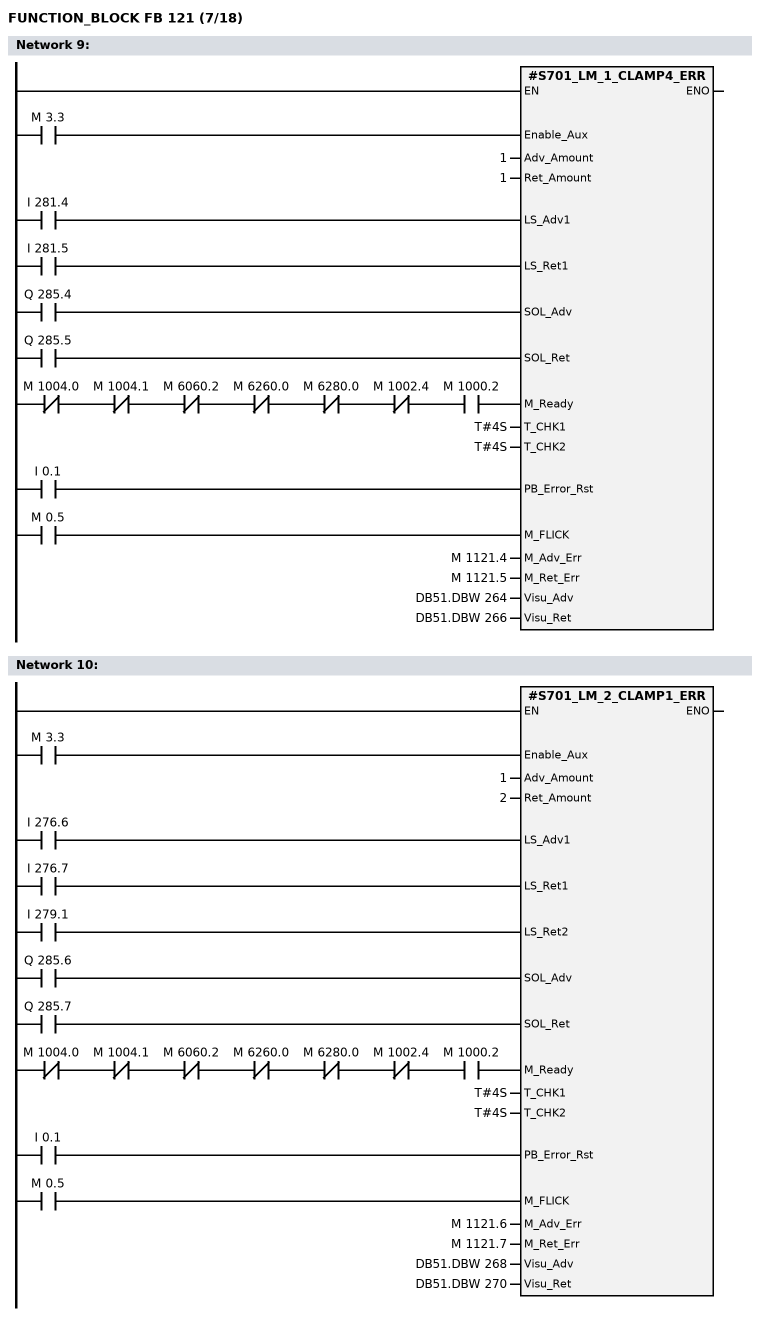

      A     M      3.3;
      =     L      0.0;
      BLD   103;
      A     I    281.4;
      =     L      0.1;
      BLD   103;
      A     I    281.5;
      =     L      0.2;
      BLD   103;
      A     Q    285.4;
      =     L      1.1;
      BLD   103;
      A     Q    285.5;
      =     L      1.2;
      BLD   103;
      AN    M   1004.0;
      AN    M   1004.1;
      AN    M   6060.2;
      AN    M   6260.0;
      AN    M   6280.0;
      AN    M   1002.4;
      A     M   1000.2;
      =     L      1.3;
      BLD   103;
      A     I      0.1;
      =     L      1.5;
      BLD   103;
      A     M      0.5;
      =     L      1.6;
      BLD   103;
      CALL #S701_LM_1_CLAMP4_ERR (
           Enable_Aux               := L      0.0,
           Adv_Amount               := 1,
           Ret_Amount               := 1,
           LS_Adv1                  := L      0.1,
           LS_Ret1                  := L      0.2,
           SOL_Adv                  := L      1.1,
           SOL_Ret                  := L      1.2,
           M_Ready                  := L      1.3,
           T_CHK1                   := T#4S,
           T_CHK2                   := T#4S,
           PB_Error_Rst             := L      1.5,
           M_FLICK                  := L      1.6,
           M_Adv_Err                := M   1121.4,
           M_Ret_Err                := M   1121.5,
           Visu_Adv                 := DB51.DBW  264,
           Visu_Ret                 := DB51.DBW  266);
      NOP   0;
NETWORK
TITLE =

      A     M      3.3;
      =     L      0.0;
      BLD   103;
      A     I    276.6;
      =     L      0.1;
      BLD   103;
      A     I    276.7;
      =     L      0.2;
      BLD   103;
      A     I    279.1;
      =     L      0.4;
      BLD   103;
      A     Q    285.6;
      =     L      1.1;
      BLD   103;
      A     Q    285.7;
      =     L      1.2;
      BLD   103;
      AN    M   1004.0;
      AN    M   1004.1;
      AN    M   6060.2;
      AN    M   6260.0;
      AN    M   6280.0;
      AN    M   1002.4;
      A     M   1000.2;
      =     L      1.3;
      BLD   103;
      A     I      0.1;
      =     L      1.5;
      BLD   103;
      A     M      0.5;
      =     L      1.6;
      BLD   103;
      CALL #S701_LM_2_CLAMP1_ERR (
           Enable_Aux               := L      0.0,
           Adv_Amount               := 1,
           Ret_Amount               := 2,
           LS_Adv1                  := L      0.1,
           LS_Ret1                  := L      0.2,
           LS_Ret2                  := L      0.4,
           SOL_Adv                  := L      1.1,
           SOL_Ret                  := L      1.2,
           M_Ready                  := L      1.3,
           T_CHK1                   := T#4S,
           T_CHK2                   := T#4S,
           PB_Error_Rst             := L      1.5,
           M_FLICK                  := L      1.6,
           M_Adv_Err                := M   1121.6,
           M_Ret_Err                := M   1121.7,
           Visu_Adv                 := DB51.DBW  268,
           Visu_Ret                 := DB51.DBW  270);
      NOP   0;
NETWORK
TITLE =
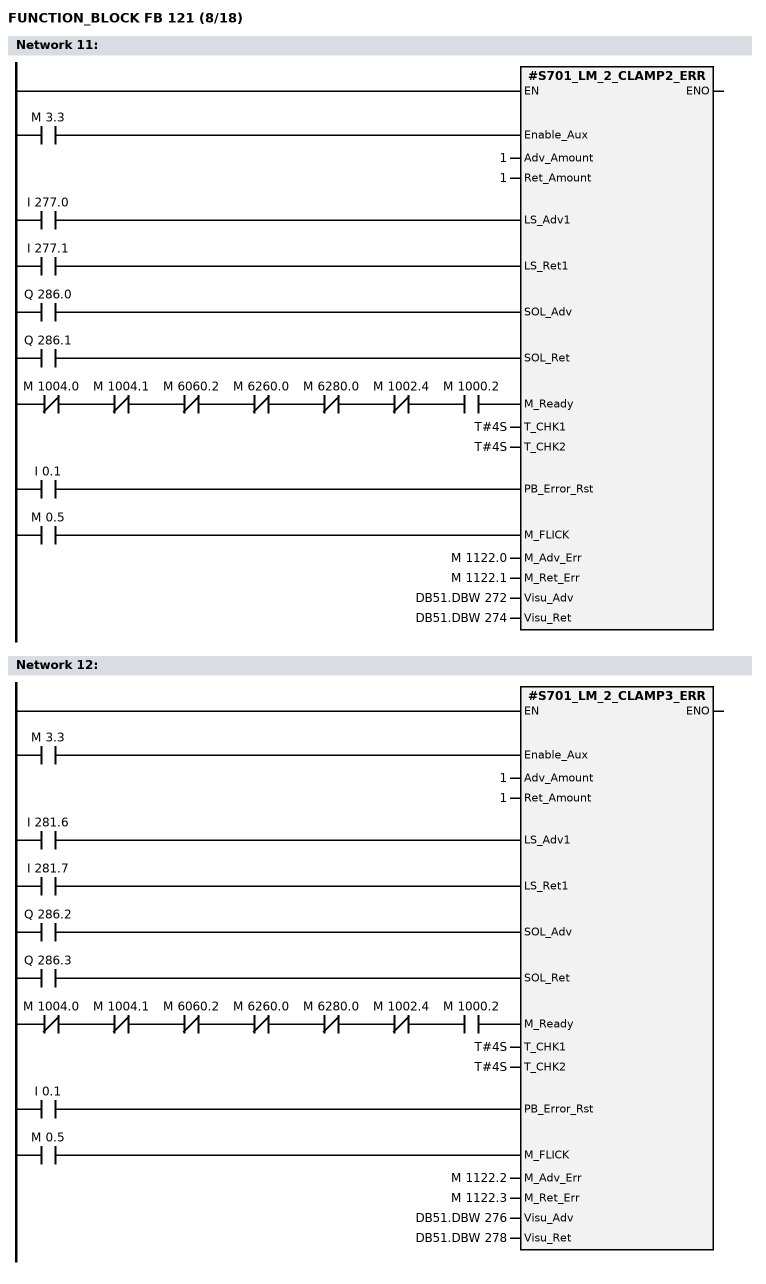

      A     M      3.3;
      =     L      0.0;
      BLD   103;
      A     I    277.0;
      =     L      0.1;
      BLD   103;
      A     I    277.1;
      =     L      0.2;
      BLD   103;
      A     Q    286.0;
      =     L      1.1;
      BLD   103;
      A     Q    286.1;
      =     L      1.2;
      BLD   103;
      AN    M   1004.0;
      AN    M   1004.1;
      AN    M   6060.2;
      AN    M   6260.0;
      AN    M   6280.0;
      AN    M   1002.4;
      A     M   1000.2;
      =     L      1.3;
      BLD   103;
      A     I      0.1;
      =     L      1.5;
      BLD   103;
      A     M      0.5;
      =     L      1.6;
      BLD   103;
      CALL #S701_LM_2_CLAMP2_ERR (
           Enable_Aux               := L      0.0,
           Adv_Amount               := 1,
           Ret_Amount               := 1,
           LS_Adv1                  := L      0.1,
           LS_Ret1                  := L      0.2,
           SOL_Adv                  := L      1.1,
           SOL_Ret                  := L      1.2,
           M_Ready                  := L      1.3,
           T_CHK1                   := T#4S,
           T_CHK2                   := T#4S,
           PB_Error_Rst             := L      1.5,
           M_FLICK                  := L      1.6,
           M_Adv_Err                := M   1122.0,
           M_Ret_Err                := M   1122.1,
           Visu_Adv                 := DB51.DBW  272,
           Visu_Ret                 := DB51.DBW  274);
      NOP   0;
NETWORK
TITLE =

      A     M      3.3;
      =     L      0.0;
      BLD   103;
      A     I    281.6;
      =     L      0.1;
      BLD   103;
      A     I    281.7;
      =     L      0.2;
      BLD   103;
      A     Q    286.2;
      =     L      1.1;
      BLD   103;
      A     Q    286.3;
      =     L      1.2;
      BLD   103;
      AN    M   1004.0;
      AN    M   1004.1;
      AN    M   6060.2;
      AN    M   6260.0;
      AN    M   6280.0;
      AN    M   1002.4;
      A     M   1000.2;
      =     L      1.3;
      BLD   103;
      A     I      0.1;
      =     L      1.5;
      BLD   103;
      A     M      0.5;
      =     L      1.6;
      BLD   103;
      CALL #S701_LM_2_CLAMP3_ERR (
           Enable_Aux               := L      0.0,
           Adv_Amount               := 1,
           Ret_Amount               := 1,
           LS_Adv1                  := L      0.1,
           LS_Ret1                  := L      0.2,
           SOL_Adv                  := L      1.1,
           SOL_Ret                  := L      1.2,
           M_Ready                  := L      1.3,
           T_CHK1                   := T#4S,
           T_CHK2                   := T#4S,
           PB_Error_Rst             := L      1.5,
           M_FLICK                  := L      1.6,
           M_Adv_Err                := M   1122.2,
           M_Ret_Err                := M   1122.3,
           Visu_Adv                 := DB51.DBW  276,
           Visu_Ret                 := DB51.DBW  278);
      NOP   0;
NETWORK
TITLE =
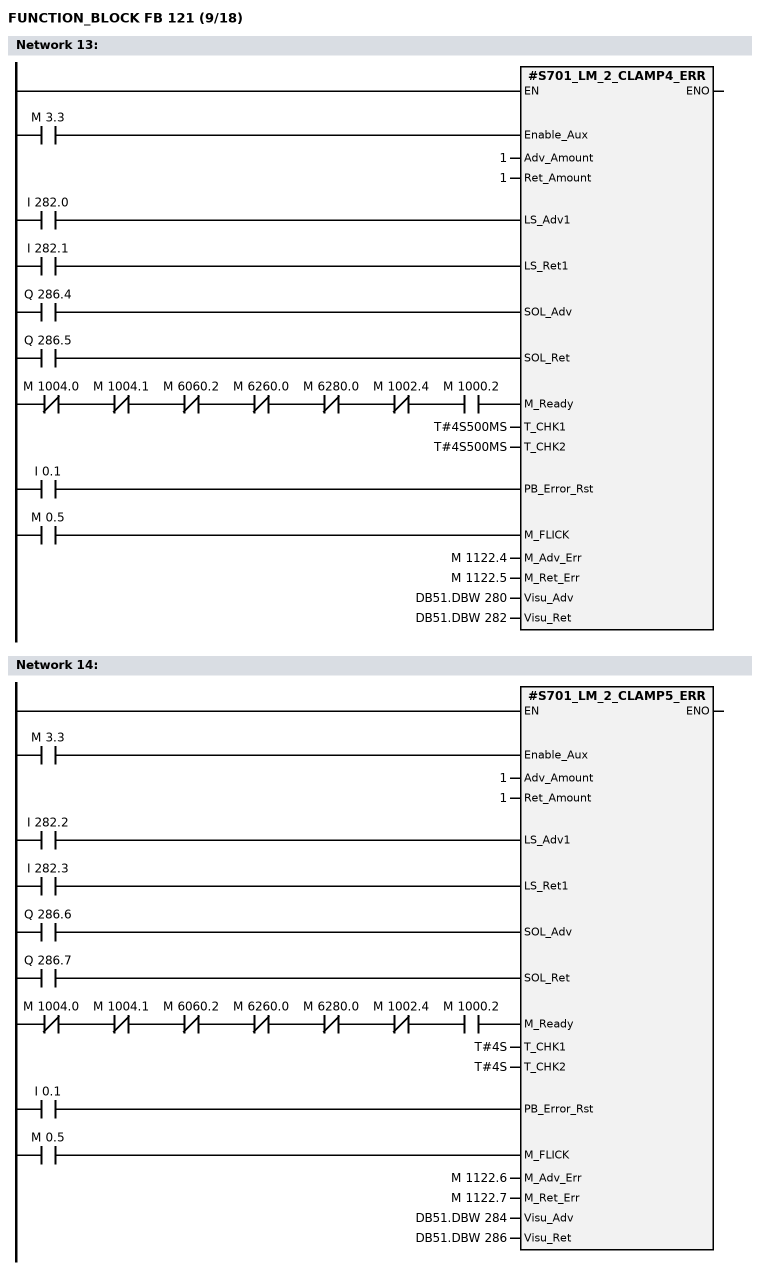

      A     M      3.3;
      =     L      0.0;
      BLD   103;
      A     I    282.0;
      =     L      0.1;
      BLD   103;
      A     I    282.1;
      =     L      0.2;
      BLD   103;
      A     Q    286.4;
      =     L      1.1;
      BLD   103;
      A     Q    286.5;
      =     L      1.2;
      BLD   103;
      AN    M   1004.0;
      AN    M   1004.1;
      AN    M   6060.2;
      AN    M   6260.0;
      AN    M   6280.0;
      AN    M   1002.4;
      A     M   1000.2;
      =     L      1.3;
      BLD   103;
      A     I      0.1;
      =     L      1.5;
      BLD   103;
      A     M      0.5;
      =     L      1.6;
      BLD   103;
      CALL #S701_LM_2_CLAMP4_ERR (
           Enable_Aux               := L      0.0,
           Adv_Amount               := 1,
           Ret_Amount               := 1,
           LS_Adv1                  := L      0.1,
           LS_Ret1                  := L      0.2,
           SOL_Adv                  := L      1.1,
           SOL_Ret                  := L      1.2,
           M_Ready                  := L      1.3,
           T_CHK1                   := T#4S500MS,
           T_CHK2                   := T#4S500MS,
           PB_Error_Rst             := L      1.5,
           M_FLICK                  := L      1.6,
           M_Adv_Err                := M   1122.4,
           M_Ret_Err                := M   1122.5,
           Visu_Adv                 := DB51.DBW  280,
           Visu_Ret                 := DB51.DBW  282);
      NOP   0;
NETWORK
TITLE =

      A     M      3.3;
      =     L      0.0;
      BLD   103;
      A     I    282.2;
      =     L      0.1;
      BLD   103;
      A     I    282.3;
      =     L      0.2;
      BLD   103;
      A     Q    286.6;
      =     L      1.1;
      BLD   103;
      A     Q    286.7;
      =     L      1.2;
      BLD   103;
      AN    M   1004.0;
      AN    M   1004.1;
      AN    M   6060.2;
      AN    M   6260.0;
      AN    M   6280.0;
      AN    M   1002.4;
      A     M   1000.2;
      =     L      1.3;
      BLD   103;
      A     I      0.1;
      =     L      1.5;
      BLD   103;
      A     M      0.5;
      =     L      1.6;
      BLD   103;
      CALL #S701_LM_2_CLAMP5_ERR (
           Enable_Aux               := L      0.0,
           Adv_Amount               := 1,
           Ret_Amount               := 1,
           LS_Adv1                  := L      0.1,
           LS_Ret1                  := L      0.2,
           SOL_Adv                  := L      1.1,
           SOL_Ret                  := L      1.2,
           M_Ready                  := L      1.3,
           T_CHK1                   := T#4S,
           T_CHK2                   := T#4S,
           PB_Error_Rst             := L      1.5,
           M_FLICK                  := L      1.6,
           M_Adv_Err                := M   1122.6,
           M_Ret_Err                := M   1122.7,
           Visu_Adv                 := DB51.DBW  284,
           Visu_Ret                 := DB51.DBW  286);
      NOP   0;
NETWORK
TITLE =
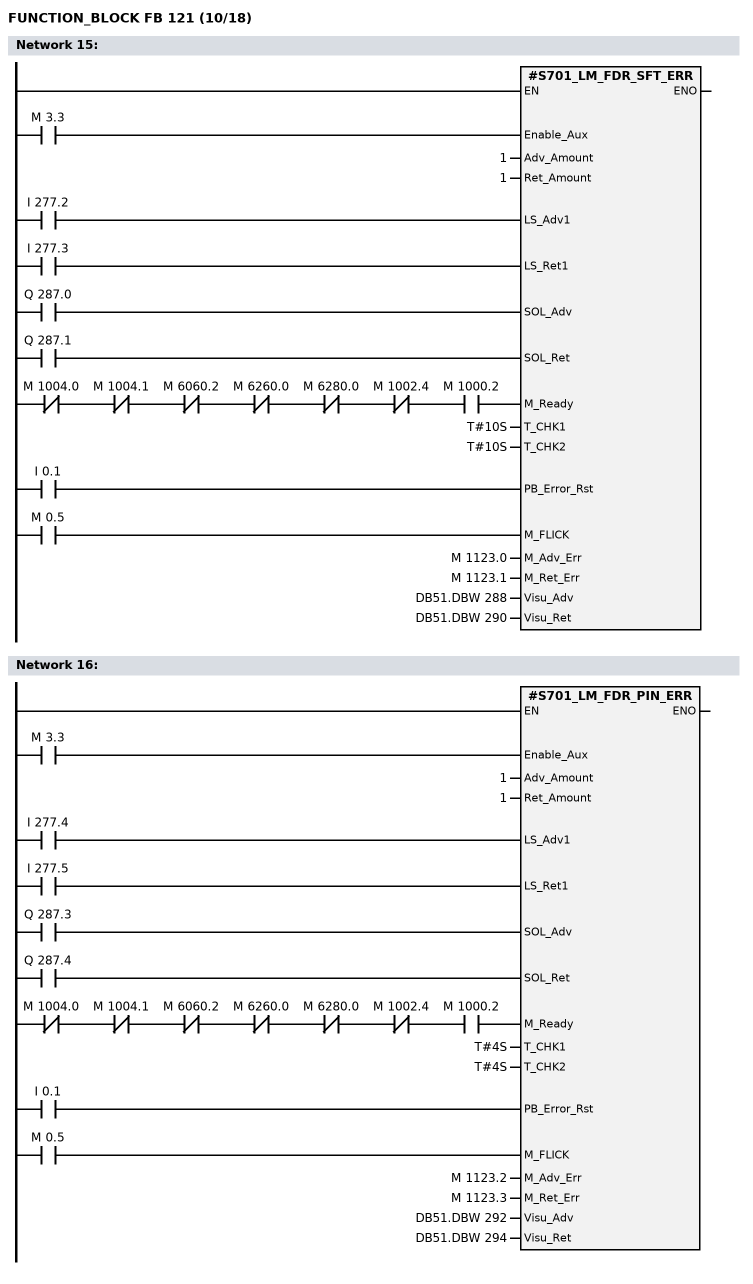

      A     M      3.3;
      =     L      0.0;
      BLD   103;
      A     I    277.2;
      =     L      0.1;
      BLD   103;
      A     I    277.3;
      =     L      0.2;
      BLD   103;
      A     Q    287.0;
      =     L      1.1;
      BLD   103;
      A     Q    287.1;
      =     L      1.2;
      BLD   103;
      AN    M   1004.0;
      AN    M   1004.1;
      AN    M   6060.2;
      AN    M   6260.0;
      AN    M   6280.0;
      AN    M   1002.4;
      A     M   1000.2;
      =     L      1.3;
      BLD   103;
      A     I      0.1;
      =     L      1.5;
      BLD   103;
      A     M      0.5;
      =     L      1.6;
      BLD   103;
      CALL #S701_LM_FDR_SFT_ERR (
           Enable_Aux               := L      0.0,
           Adv_Amount               := 1,
           Ret_Amount               := 1,
           LS_Adv1                  := L      0.1,
           LS_Ret1                  := L      0.2,
           SOL_Adv                  := L      1.1,
           SOL_Ret                  := L      1.2,
           M_Ready                  := L      1.3,
           T_CHK1                   := T#10S,
           T_CHK2                   := T#10S,
           PB_Error_Rst             := L      1.5,
           M_FLICK                  := L      1.6,
           M_Adv_Err                := M   1123.0,
           M_Ret_Err                := M   1123.1,
           Visu_Adv                 := DB51.DBW  288,
           Visu_Ret                 := DB51.DBW  290);
      NOP   0;
NETWORK
TITLE =

      A     M      3.3;
      =     L      0.0;
      BLD   103;
      A     I    277.4;
      =     L      0.1;
      BLD   103;
      A     I    277.5;
      =     L      0.2;
      BLD   103;
      A     Q    287.3;
      =     L      1.1;
      BLD   103;
      A     Q    287.4;
      =     L      1.2;
      BLD   103;
      AN    M   1004.0;
      AN    M   1004.1;
      AN    M   6060.2;
      AN    M   6260.0;
      AN    M   6280.0;
      AN    M   1002.4;
      A     M   1000.2;
      =     L      1.3;
      BLD   103;
      A     I      0.1;
      =     L      1.5;
      BLD   103;
      A     M      0.5;
      =     L      1.6;
      BLD   103;
      CALL #S701_LM_FDR_PIN_ERR (
           Enable_Aux               := L      0.0,
           Adv_Amount               := 1,
           Ret_Amount               := 1,
           LS_Adv1                  := L      0.1,
           LS_Ret1                  := L      0.2,
           SOL_Adv                  := L      1.1,
           SOL_Ret                  := L      1.2,
           M_Ready                  := L      1.3,
           T_CHK1                   := T#4S,
           T_CHK2                   := T#4S,
           PB_Error_Rst             := L      1.5,
           M_FLICK                  := L      1.6,
           M_Adv_Err                := M   1123.2,
           M_Ret_Err                := M   1123.3,
           Visu_Adv                 := DB51.DBW  292,
           Visu_Ret                 := DB51.DBW  294);
      NOP   0;
NETWORK
TITLE =
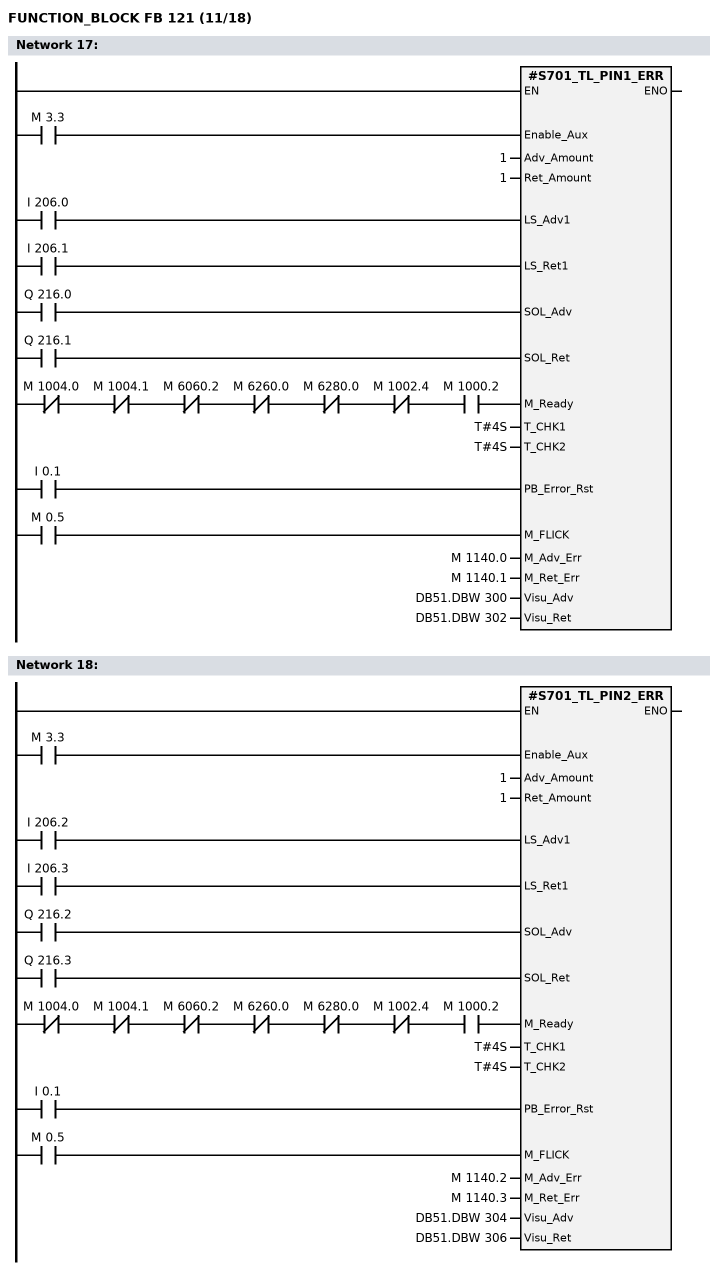

      A     M      3.3;
      =     L      0.0;
      BLD   103;
      A     I    206.0;
      =     L      0.1;
      BLD   103;
      A     I    206.1;
      =     L      0.2;
      BLD   103;
      A     Q    216.0;
      =     L      1.1;
      BLD   103;
      A     Q    216.1;
      =     L      1.2;
      BLD   103;
      AN    M   1004.0;
      AN    M   1004.1;
      AN    M   6060.2;
      AN    M   6260.0;
      AN    M   6280.0;
      AN    M   1002.4;
      A     M   1000.2;
      =     L      1.3;
      BLD   103;
      A     I      0.1;
      =     L      1.5;
      BLD   103;
      A     M      0.5;
      =     L      1.6;
      BLD   103;
      CALL #S701_TL_PIN1_ERR (
           Enable_Aux               := L      0.0,
           Adv_Amount               := 1,
           Ret_Amount               := 1,
           LS_Adv1                  := L      0.1,
           LS_Ret1                  := L      0.2,
           SOL_Adv                  := L      1.1,
           SOL_Ret                  := L      1.2,
           M_Ready                  := L      1.3,
           T_CHK1                   := T#4S,
           T_CHK2                   := T#4S,
           PB_Error_Rst             := L      1.5,
           M_FLICK                  := L      1.6,
           M_Adv_Err                := M   1140.0,
           M_Ret_Err                := M   1140.1,
           Visu_Adv                 := DB51.DBW  300,
           Visu_Ret                 := DB51.DBW  302);
      NOP   0;
NETWORK
TITLE =

      A     M      3.3;
      =     L      0.0;
      BLD   103;
      A     I    206.2;
      =     L      0.1;
      BLD   103;
      A     I    206.3;
      =     L      0.2;
      BLD   103;
      A     Q    216.2;
      =     L      1.1;
      BLD   103;
      A     Q    216.3;
      =     L      1.2;
      BLD   103;
      AN    M   1004.0;
      AN    M   1004.1;
      AN    M   6060.2;
      AN    M   6260.0;
      AN    M   6280.0;
      AN    M   1002.4;
      A     M   1000.2;
      =     L      1.3;
      BLD   103;
      A     I      0.1;
      =     L      1.5;
      BLD   103;
      A     M      0.5;
      =     L      1.6;
      BLD   103;
      CALL #S701_TL_PIN2_ERR (
           Enable_Aux               := L      0.0,
           Adv_Amount               := 1,
           Ret_Amount               := 1,
           LS_Adv1                  := L      0.1,
           LS_Ret1                  := L      0.2,
           SOL_Adv                  := L      1.1,
           SOL_Ret                  := L      1.2,
           M_Ready                  := L      1.3,
           T_CHK1                   := T#4S,
           T_CHK2                   := T#4S,
           PB_Error_Rst             := L      1.5,
           M_FLICK                  := L      1.6,
           M_Adv_Err                := M   1140.2,
           M_Ret_Err                := M   1140.3,
           Visu_Adv                 := DB51.DBW  304,
           Visu_Ret                 := DB51.DBW  306);
      NOP   0;
NETWORK
TITLE =
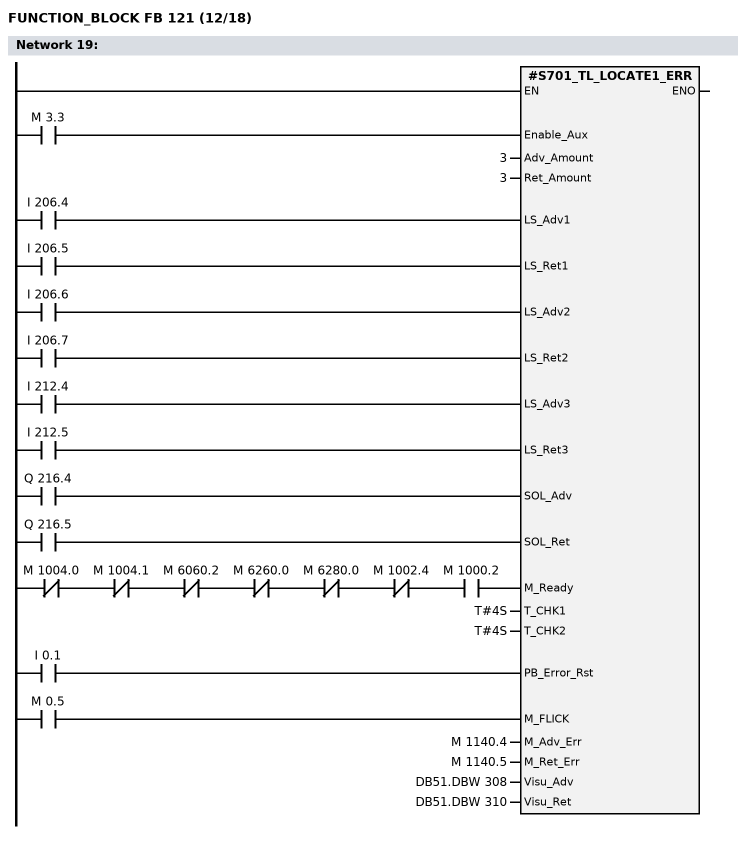

      A     M      3.3;
      =     L      0.0;
      BLD   103;
      A     I    206.4;
      =     L      0.1;
      BLD   103;
      A     I    206.5;
      =     L      0.2;
      BLD   103;
      A     I    206.6;
      =     L      0.3;
      BLD   103;
      A     I    206.7;
      =     L      0.4;
      BLD   103;
      A     I    212.4;
      =     L      0.5;
      BLD   103;
      A     I    212.5;
      =     L      0.6;
      BLD   103;
      A     Q    216.4;
      =     L      1.1;
      BLD   103;
      A     Q    216.5;
      =     L      1.2;
      BLD   103;
      AN    M   1004.0;
      AN    M   1004.1;
      AN    M   6060.2;
      AN    M   6260.0;
      AN    M   6280.0;
      AN    M   1002.4;
      A     M   1000.2;
      =     L      1.3;
      BLD   103;
      A     I      0.1;
      =     L      1.5;
      BLD   103;
      A     M      0.5;
      =     L      1.6;
      BLD   103;
      CALL #S701_TL_LOCATE1_ERR (
           Enable_Aux               := L      0.0,
           Adv_Amount               := 3,
           Ret_Amount               := 3,
           LS_Adv1                  := L      0.1,
           LS_Ret1                  := L      0.2,
           LS_Adv2                  := L      0.3,
           LS_Ret2                  := L      0.4,
           LS_Adv3                  := L      0.5,
           LS_Ret3                  := L      0.6,
           SOL_Adv                  := L      1.1,
           SOL_Ret                  := L      1.2,
           M_Ready                  := L      1.3,
           T_CHK1                   := T#4S,
           T_CHK2                   := T#4S,
           PB_Error_Rst             := L      1.5,
           M_FLICK                  := L      1.6,
           M_Adv_Err                := M   1140.4,
           M_Ret_Err                := M   1140.5,
           Visu_Adv                 := DB51.DBW  308,
           Visu_Ret                 := DB51.DBW  310);
      NOP   0;
NETWORK
TITLE =
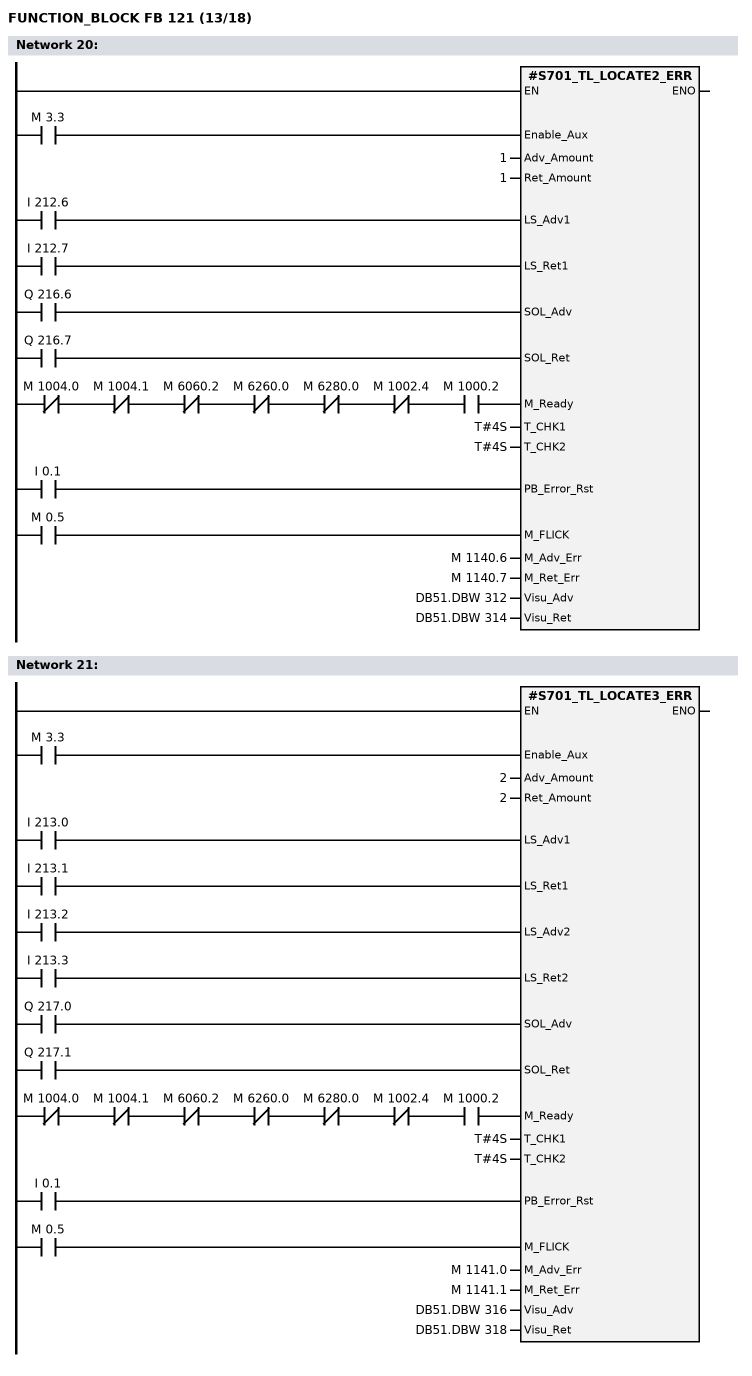

      A     M      3.3;
      =     L      0.0;
      BLD   103;
      A     I    212.6;
      =     L      0.1;
      BLD   103;
      A     I    212.7;
      =     L      0.2;
      BLD   103;
      A     Q    216.6;
      =     L      1.1;
      BLD   103;
      A     Q    216.7;
      =     L      1.2;
      BLD   103;
      AN    M   1004.0;
      AN    M   1004.1;
      AN    M   6060.2;
      AN    M   6260.0;
      AN    M   6280.0;
      AN    M   1002.4;
      A     M   1000.2;
      =     L      1.3;
      BLD   103;
      A     I      0.1;
      =     L      1.5;
      BLD   103;
      A     M      0.5;
      =     L      1.6;
      BLD   103;
      CALL #S701_TL_LOCATE2_ERR (
           Enable_Aux               := L      0.0,
           Adv_Amount               := 1,
           Ret_Amount               := 1,
           LS_Adv1                  := L      0.1,
           LS_Ret1                  := L      0.2,
           SOL_Adv                  := L      1.1,
           SOL_Ret                  := L      1.2,
           M_Ready                  := L      1.3,
           T_CHK1                   := T#4S,
           T_CHK2                   := T#4S,
           PB_Error_Rst             := L      1.5,
           M_FLICK                  := L      1.6,
           M_Adv_Err                := M   1140.6,
           M_Ret_Err                := M   1140.7,
           Visu_Adv                 := DB51.DBW  312,
           Visu_Ret                 := DB51.DBW  314);
      NOP   0;
NETWORK
TITLE =

      A     M      3.3;
      =     L      0.0;
      BLD   103;
      A     I    213.0;
      =     L      0.1;
      BLD   103;
      A     I    213.1;
      =     L      0.2;
      BLD   103;
      A     I    213.2;
      =     L      0.3;
      BLD   103;
      A     I    213.3;
      =     L      0.4;
      BLD   103;
      A     Q    217.0;
      =     L      1.1;
      BLD   103;
      A     Q    217.1;
      =     L      1.2;
      BLD   103;
      AN    M   1004.0;
      AN    M   1004.1;
      AN    M   6060.2;
      AN    M   6260.0;
      AN    M   6280.0;
      AN    M   1002.4;
      A     M   1000.2;
      =     L      1.3;
      BLD   103;
      A     I      0.1;
      =     L      1.5;
      BLD   103;
      A     M      0.5;
      =     L      1.6;
      BLD   103;
      CALL #S701_TL_LOCATE3_ERR (
           Enable_Aux               := L      0.0,
           Adv_Amount               := 2,
           Ret_Amount               := 2,
           LS_Adv1                  := L      0.1,
           LS_Ret1                  := L      0.2,
           LS_Adv2                  := L      0.3,
           LS_Ret2                  := L      0.4,
           SOL_Adv                  := L      1.1,
           SOL_Ret                  := L      1.2,
           M_Ready                  := L      1.3,
           T_CHK1                   := T#4S,
           T_CHK2                   := T#4S,
           PB_Error_Rst             := L      1.5,
           M_FLICK                  := L      1.6,
           M_Adv_Err                := M   1141.0,
           M_Ret_Err                := M   1141.1,
           Visu_Adv                 := DB51.DBW  316,
           Visu_Ret                 := DB51.DBW  318);
      NOP   0;
NETWORK
TITLE =
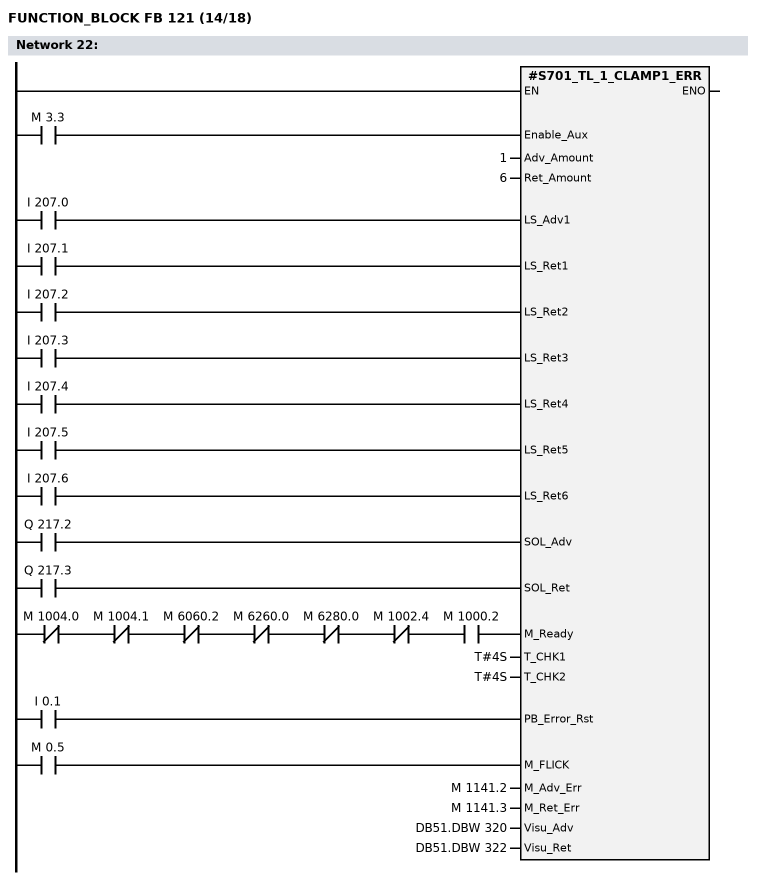

      A     M      3.3;
      =     L      0.0;
      BLD   103;
      A     I    207.0;
      =     L      0.1;
      BLD   103;
      A     I    207.1;
      =     L      0.2;
      BLD   103;
      A     I    207.2;
      =     L      0.4;
      BLD   103;
      A     I    207.3;
      =     L      0.6;
      BLD   103;
      A     I    207.4;
      =     L      1.0;
      BLD   103;
      A     I    207.5;
      =     L      1.2;
      BLD   103;
      A     I    207.6;
      =     L      1.4;
      BLD   103;
      A     Q    217.2;
      =     L      2.1;
      BLD   103;
      A     Q    217.3;
      =     L      2.2;
      BLD   103;
      AN    M   1004.0;
      AN    M   1004.1;
      AN    M   6060.2;
      AN    M   6260.0;
      AN    M   6280.0;
      AN    M   1002.4;
      A     M   1000.2;
      =     L      2.3;
      BLD   103;
      A     I      0.1;
      =     L      2.5;
      BLD   103;
      A     M      0.5;
      =     L      2.6;
      BLD   103;
      CALL #S701_TL_1_CLAMP1_ERR (
           Enable_Aux               := L      0.0,
           Adv_Amount               := 1,
           Ret_Amount               := 6,
           LS_Adv1                  := L      0.1,
           LS_Ret1                  := L      0.2,
           LS_Ret2                  := L      0.4,
           LS_Ret3                  := L      0.6,
           LS_Ret4                  := L      1.0,
           LS_Ret5                  := L      1.2,
           LS_Ret6                  := L      1.4,
           SOL_Adv                  := L      2.1,
           SOL_Ret                  := L      2.2,
           M_Ready                  := L      2.3,
           T_CHK1                   := T#4S,
           T_CHK2                   := T#4S,
           PB_Error_Rst             := L      2.5,
           M_FLICK                  := L      2.6,
           M_Adv_Err                := M   1141.2,
           M_Ret_Err                := M   1141.3,
           Visu_Adv                 := DB51.DBW  320,
           Visu_Ret                 := DB51.DBW  322);
      NOP   0;
NETWORK
TITLE =
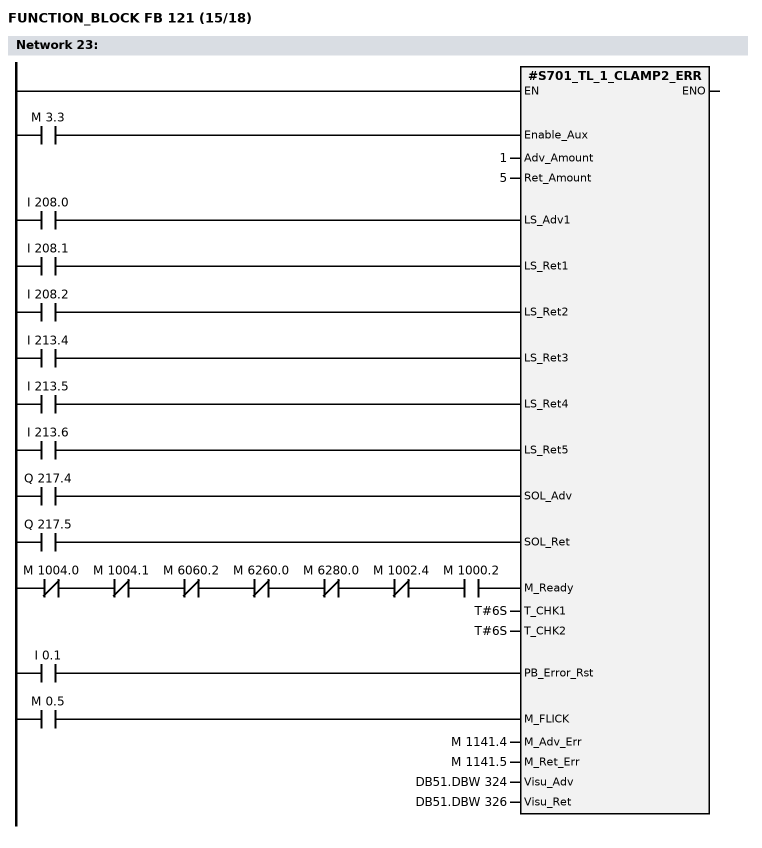

      A     M      3.3;
      =     L      0.0;
      BLD   103;
      A     I    208.0;
      =     L      0.1;
      BLD   103;
      A     I    208.1;
      =     L      0.2;
      BLD   103;
      A     I    208.2;
      =     L      0.4;
      BLD   103;
      A     I    213.4;
      =     L      0.6;
      BLD   103;
      A     I    213.5;
      =     L      1.0;
      BLD   103;
      A     I    213.6;
      =     L      1.2;
      BLD   103;
      A     Q    217.4;
      =     L      2.1;
      BLD   103;
      A     Q    217.5;
      =     L      2.2;
      BLD   103;
      AN    M   1004.0;
      AN    M   1004.1;
      AN    M   6060.2;
      AN    M   6260.0;
      AN    M   6280.0;
      AN    M   1002.4;
      A     M   1000.2;
      =     L      2.3;
      BLD   103;
      A     I      0.1;
      =     L      2.5;
      BLD   103;
      A     M      0.5;
      =     L      2.6;
      BLD   103;
      CALL #S701_TL_1_CLAMP2_ERR (
           Enable_Aux               := L      0.0,
           Adv_Amount               := 1,
           Ret_Amount               := 5,
           LS_Adv1                  := L      0.1,
           LS_Ret1                  := L      0.2,
           LS_Ret2                  := L      0.4,
           LS_Ret3                  := L      0.6,
           LS_Ret4                  := L      1.0,
           LS_Ret5                  := L      1.2,
           SOL_Adv                  := L      2.1,
           SOL_Ret                  := L      2.2,
           M_Ready                  := L      2.3,
           T_CHK1                   := T#6S,
           T_CHK2                   := T#6S,
           PB_Error_Rst             := L      2.5,
           M_FLICK                  := L      2.6,
           M_Adv_Err                := M   1141.4,
           M_Ret_Err                := M   1141.5,
           Visu_Adv                 := DB51.DBW  324,
           Visu_Ret                 := DB51.DBW  326);
      NOP   0;
NETWORK
TITLE =
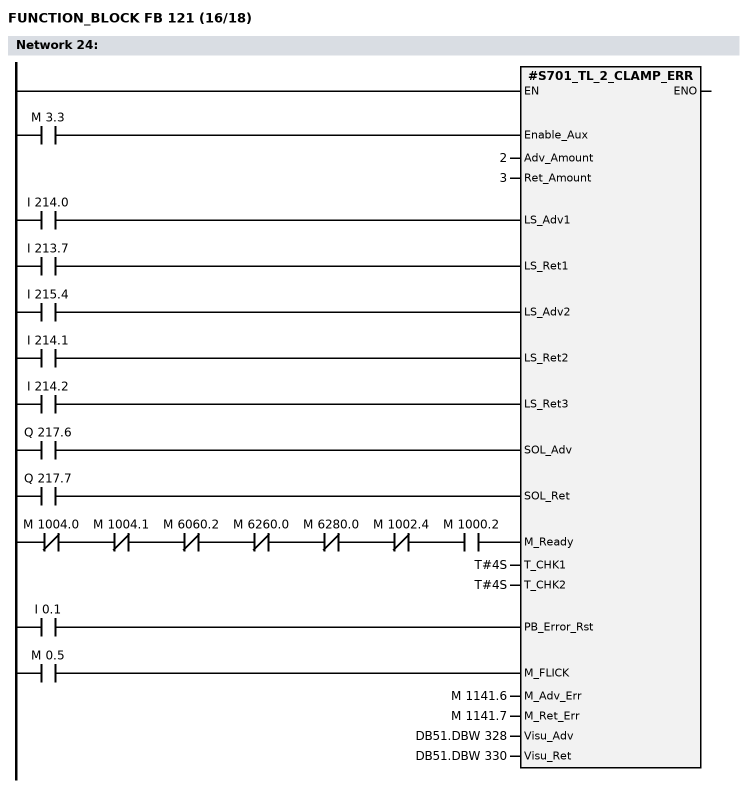

      A     M      3.3;
      =     L      0.0;
      BLD   103;
      A     I    214.0;
      =     L      0.1;
      BLD   103;
      A     I    213.7;
      =     L      0.2;
      BLD   103;
      A     I    215.4;
      =     L      0.3;
      BLD   103;
      A     I    214.1;
      =     L      0.4;
      BLD   103;
      A     I    214.2;
      =     L      0.6;
      BLD   103;
      A     Q    217.6;
      =     L      2.1;
      BLD   103;
      A     Q    217.7;
      =     L      2.2;
      BLD   103;
      AN    M   1004.0;
      AN    M   1004.1;
      AN    M   6060.2;
      AN    M   6260.0;
      AN    M   6280.0;
      AN    M   1002.4;
      A     M   1000.2;
      =     L      2.3;
      BLD   103;
      A     I      0.1;
      =     L      2.5;
      BLD   103;
      A     M      0.5;
      =     L      2.6;
      BLD   103;
      CALL #S701_TL_2_CLAMP_ERR (
           Enable_Aux               := L      0.0,
           Adv_Amount               := 2,
           Ret_Amount               := 3,
           LS_Adv1                  := L      0.1,
           LS_Ret1                  := L      0.2,
           LS_Adv2                  := L      0.3,
           LS_Ret2                  := L      0.4,
           LS_Ret3                  := L      0.6,
           SOL_Adv                  := L      2.1,
           SOL_Ret                  := L      2.2,
           M_Ready                  := L      2.3,
           T_CHK1                   := T#4S,
           T_CHK2                   := T#4S,
           PB_Error_Rst             := L      2.5,
           M_FLICK                  := L      2.6,
           M_Adv_Err                := M   1141.6,
           M_Ret_Err                := M   1141.7,
           Visu_Adv                 := DB51.DBW  328,
           Visu_Ret                 := DB51.DBW  330);
      NOP   0;
NETWORK
TITLE =
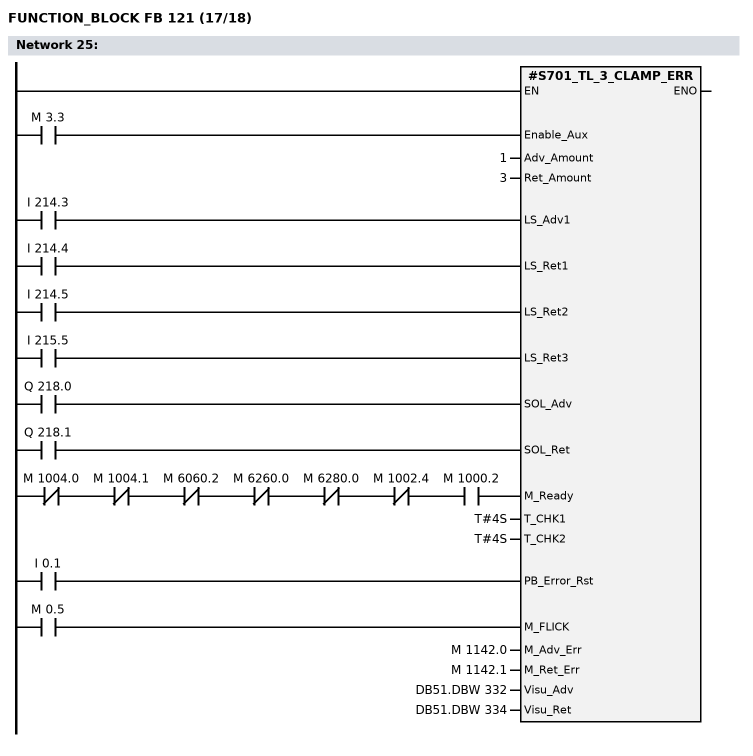

      A     M      3.3;
      =     L      0.0;
      BLD   103;
      A     I    214.3;
      =     L      0.1;
      BLD   103;
      A     I    214.4;
      =     L      0.2;
      BLD   103;
      A     I    214.5;
      =     L      0.4;
      BLD   103;
      A     I    215.5;
      =     L      0.6;
      BLD   103;
      A     Q    218.0;
      =     L      2.1;
      BLD   103;
      A     Q    218.1;
      =     L      2.2;
      BLD   103;
      AN    M   1004.0;
      AN    M   1004.1;
      AN    M   6060.2;
      AN    M   6260.0;
      AN    M   6280.0;
      AN    M   1002.4;
      A     M   1000.2;
      =     L      2.3;
      BLD   103;
      A     I      0.1;
      =     L      2.5;
      BLD   103;
      A     M      0.5;
      =     L      2.6;
      BLD   103;
      CALL #S701_TL_3_CLAMP_ERR (
           Enable_Aux               := L      0.0,
           Adv_Amount               := 1,
           Ret_Amount               := 3,
           LS_Adv1                  := L      0.1,
           LS_Ret1                  := L      0.2,
           LS_Ret2                  := L      0.4,
           LS_Ret3                  := L      0.6,
           SOL_Adv                  := L      2.1,
           SOL_Ret                  := L      2.2,
           M_Ready                  := L      2.3,
           T_CHK1                   := T#4S,
           T_CHK2                   := T#4S,
           PB_Error_Rst             := L      2.5,
           M_FLICK                  := L      2.6,
           M_Adv_Err                := M   1142.0,
           M_Ret_Err                := M   1142.1,
           Visu_Adv                 := DB51.DBW  332,
           Visu_Ret                 := DB51.DBW  334);
      NOP   0;
NETWORK
TITLE =
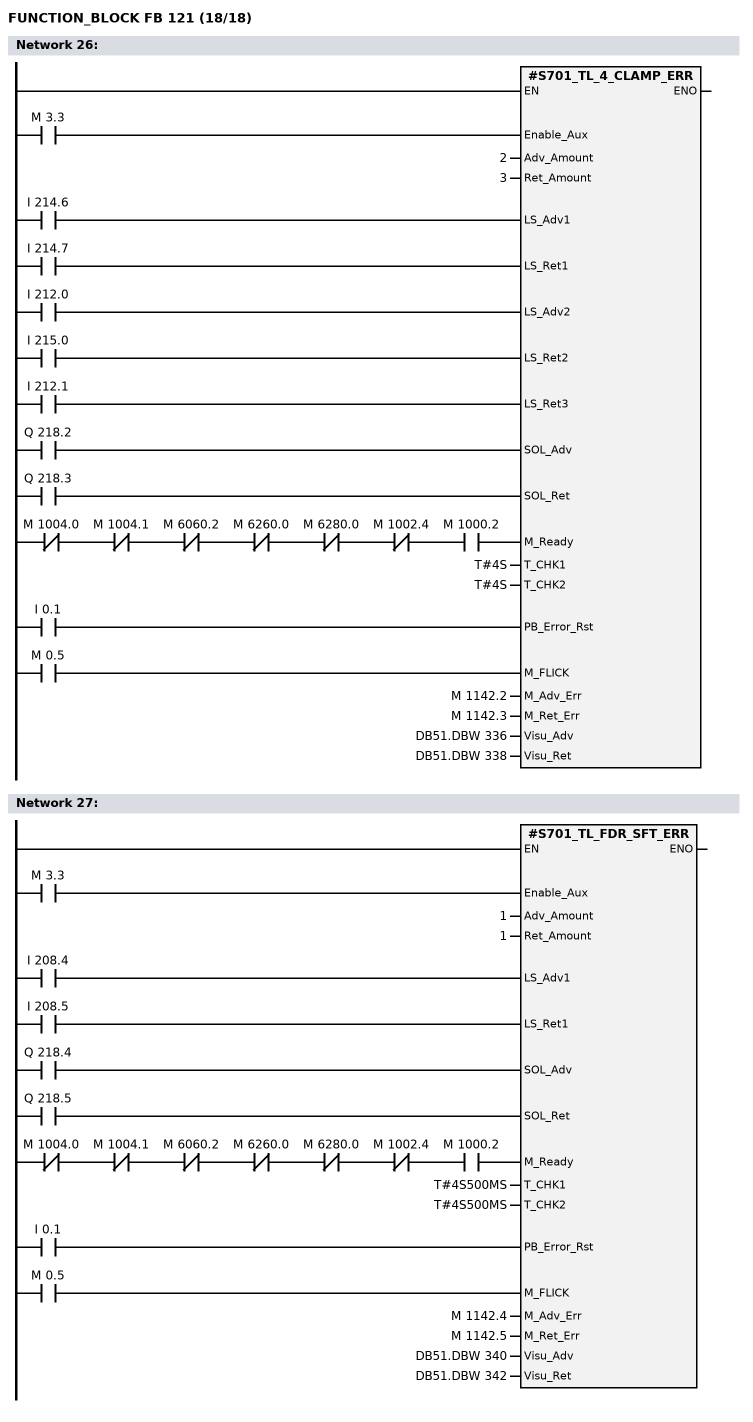

      A     M      3.3;
      =     L      0.0;
      BLD   103;
      A     I    214.6;
      =     L      0.1;
      BLD   103;
      A     I    214.7;
      =     L      0.2;
      BLD   103;
      A     I    212.0;
      =     L      0.3;
      BLD   103;
      A     I    215.0;
      =     L      0.4;
      BLD   103;
      A     I    212.1;
      =     L      0.6;
      BLD   103;
      A     Q    218.2;
      =     L      2.1;
      BLD   103;
      A     Q    218.3;
      =     L      2.2;
      BLD   103;
      AN    M   1004.0;
      AN    M   1004.1;
      AN    M   6060.2;
      AN    M   6260.0;
      AN    M   6280.0;
      AN    M   1002.4;
      A     M   1000.2;
      =     L      2.3;
      BLD   103;
      A     I      0.1;
      =     L      2.5;
      BLD   103;
      A     M      0.5;
      =     L      2.6;
      BLD   103;
      CALL #S701_TL_4_CLAMP_ERR (
           Enable_Aux               := L      0.0,
           Adv_Amount               := 2,
           Ret_Amount               := 3,
           LS_Adv1                  := L      0.1,
           LS_Ret1                  := L      0.2,
           LS_Adv2                  := L      0.3,
           LS_Ret2                  := L      0.4,
           LS_Ret3                  := L      0.6,
           SOL_Adv                  := L      2.1,
           SOL_Ret                  := L      2.2,
           M_Ready                  := L      2.3,
           T_CHK1                   := T#4S,
           T_CHK2                   := T#4S,
           PB_Error_Rst             := L      2.5,
           M_FLICK                  := L      2.6,
           M_Adv_Err                := M   1142.2,
           M_Ret_Err                := M   1142.3,
           Visu_Adv                 := DB51.DBW  336,
           Visu_Ret                 := DB51.DBW  338);
      NOP   0;
NETWORK
TITLE =

      A     M      3.3;
      =     L      0.0;
      BLD   103;
      A     I    208.4;
      =     L      0.1;
      BLD   103;
      A     I    208.5;
      =     L      0.2;
      BLD   103;
      A     Q    218.4;
      =     L      2.1;
      BLD   103;
      A     Q    218.5;
      =     L      2.2;
      BLD   103;
      AN    M   1004.0;
      AN    M   1004.1;
      AN    M   6060.2;
      AN    M   6260.0;
      AN    M   6280.0;
      AN    M   1002.4;
      A     M   1000.2;
      =     L      2.3;
      BLD   103;
      A     I      0.1;
      =     L      2.5;
      BLD   103;
      A     M      0.5;
      =     L      2.6;
      BLD   103;
      CALL #S701_TL_FDR_SFT_ERR (
           Enable_Aux               := L      0.0,
           Adv_Amount               := 1,
           Ret_Amount               := 1,
           LS_Adv1                  := L      0.1,
           LS_Ret1                  := L      0.2,
           SOL_Adv                  := L      2.1,
           SOL_Ret                  := L      2.2,
           M_Ready                  := L      2.3,
           T_CHK1                   := T#4S500MS,
           T_CHK2                   := T#4S500MS,
           PB_Error_Rst             := L      2.5,
           M_FLICK                  := L      2.6,
           M_Adv_Err                := M   1142.4,
           M_Ret_Err                := M   1142.5,
           Visu_Adv                 := DB51.DBW  340,
           Visu_Ret                 := DB51.DBW  342);
      NOP   0;
END_FUNCTION_BLOCK

DATA_BLOCK DB 121
TITLE =
VERSION : 0.0

 FB 121
BEGIN
   S701_RETURN_LOCK_ERR.Enable_Aux := FALSE;
   S701_RETURN_LOCK_ERR.Adv_Amount := 0;
   S701_RETURN_LOCK_ERR.Ret_Amount := 0;
   S701_RETURN_LOCK_ERR.LS_Adv1 := FALSE;
   S701_RETURN_LOCK_ERR.LS_Ret1 := FALSE;
   S701_RETURN_LOCK_ERR.LS_Adv2 := FALSE;
   S701_RETURN_LOCK_ERR.LS_Ret2 := FALSE;
   S701_RETURN_LOCK_ERR.LS_Adv3 := FALSE;
   S701_RETURN_LOCK_ERR.LS_Ret3 := FALSE;
   S701_RETURN_LOCK_ERR.LS_Adv4 := FALSE;
   S701_RETURN_LOCK_ERR.LS_Ret4 := FALSE;
   S701_RETURN_LOCK_ERR.SOL_Adv := FALSE;
   S701_RETURN_LOCK_ERR.SOL_Ret := FALSE;
   S701_RETURN_LOCK_ERR.M_Ready := FALSE;
   S701_RETURN_LOCK_ERR.T_CHK1 := T#0MS;
   S701_RETURN_LOCK_ERR.T_CHK2 := T#0MS;
   S701_RETURN_LOCK_ERR.PB_Lamp_CHK := FALSE;
   S701_RETURN_LOCK_ERR.PB_Error_Rst := FALSE;
   S701_RETURN_LOCK_ERR.M_FLICK := FALSE;
   S701_RETURN_LOCK_ERR.M_Adv_Err := FALSE;
   S701_RETURN_LOCK_ERR.M_Ret_Err := FALSE;
   S701_RETURN_LOCK_ERR.LP_Adv := FALSE;
   S701_RETURN_LOCK_ERR.LP_Ret := FALSE;
   S701_RETURN_LOCK_ERR.Visu_Adv := W#16#0;
   S701_RETURN_LOCK_ERR.Visu_Ret := W#16#0;
   S701_RETURN_LOCK_ERR.Error_T1.IN := FALSE;
   S701_RETURN_LOCK_ERR.Error_T1.PT := T#0MS;
   S701_RETURN_LOCK_ERR.Error_T1.Q := FALSE;
   S701_RETURN_LOCK_ERR.Error_T1.ET := T#0MS;
   S701_RETURN_LOCK_ERR.Error_T1.STATE := B#16#0;
   S701_RETURN_LOCK_ERR.Error_T1.STIME := T#0MS;
   S701_RETURN_LOCK_ERR.Error_T1.ATIME := T#0MS;
   S701_RETURN_LOCK_ERR.Error_T2.IN := FALSE;
   S701_RETURN_LOCK_ERR.Error_T2.PT := T#0MS;
   S701_RETURN_LOCK_ERR.Error_T2.Q := FALSE;
   S701_RETURN_LOCK_ERR.Error_T2.ET := T#0MS;
   S701_RETURN_LOCK_ERR.Error_T2.STATE := B#16#0;
   S701_RETURN_LOCK_ERR.Error_T2.STIME := T#0MS;
   S701_RETURN_LOCK_ERR.Error_T2.ATIME := T#0MS;
   S701_RETURN_LOCK_ERR.CHK_Aux1 := FALSE;
   S701_RETURN_LOCK_ERR.CHK_Aux2 := FALSE;
   S701_RETURN_LOCK_ERR.Error_T1_DN := FALSE;
   S701_RETURN_LOCK_ERR.Error_T2_DN := FALSE;
   S701_RETURN_LOCK_ERR.Adv_Memo := FALSE;
   S701_RETURN_LOCK_ERR.Visu_Adv_Arr[0] := FALSE;
   S701_RETURN_LOCK_ERR.Visu_Adv_Arr[1] := FALSE;
   S701_RETURN_LOCK_ERR.Visu_Adv_Arr[2] := FALSE;
   S701_RETURN_LOCK_ERR.Visu_Adv_Arr[3] := FALSE;
   S701_RETURN_LOCK_ERR.Visu_Adv_Arr[4] := FALSE;
   S701_RETURN_LOCK_ERR.Visu_Adv_Arr[5] := FALSE;
   S701_RETURN_LOCK_ERR.Visu_Adv_Arr[6] := FALSE;
   S701_RETURN_LOCK_ERR.Visu_Adv_Arr[7] := FALSE;
   S701_RETURN_LOCK_ERR.Visu_Adv_Arr[8] := FALSE;
   S701_RETURN_LOCK_ERR.Visu_Adv_Arr[9] := FALSE;
   S701_RETURN_LOCK_ERR.Visu_Adv_Arr[10] := FALSE;
   S701_RETURN_LOCK_ERR.Visu_Adv_Arr[11] := FALSE;
   S701_RETURN_LOCK_ERR.Visu_Adv_Arr[12] := FALSE;
   S701_RETURN_LOCK_ERR.Visu_Adv_Arr[13] := FALSE;
   S701_RETURN_LOCK_ERR.Visu_Adv_Arr[14] := FALSE;
   S701_RETURN_LOCK_ERR.Visu_Adv_Arr[15] := FALSE;
   S701_RETURN_LOCK_ERR.Visu_Ret_Arr[0] := FALSE;
   S701_RETURN_LOCK_ERR.Visu_Ret_Arr[1] := FALSE;
   S701_RETURN_LOCK_ERR.Visu_Ret_Arr[2] := FALSE;
   S701_RETURN_LOCK_ERR.Visu_Ret_Arr[3] := FALSE;
   S701_RETURN_LOCK_ERR.Visu_Ret_Arr[4] := FALSE;
   S701_RETURN_LOCK_ERR.Visu_Ret_Arr[5] := FALSE;
   S701_RETURN_LOCK_ERR.Visu_Ret_Arr[6] := FALSE;
   S701_RETURN_LOCK_ERR.Visu_Ret_Arr[7] := FALSE;
   S701_RETURN_LOCK_ERR.Visu_Ret_Arr[8] := FALSE;
   S701_RETURN_LOCK_ERR.Visu_Ret_Arr[9] := FALSE;
   S701_RETURN_LOCK_ERR.Visu_Ret_Arr[10] := FALSE;
   S701_RETURN_LOCK_ERR.Visu_Ret_Arr[11] := FALSE;
   S701_RETURN_LOCK_ERR.Visu_Ret_Arr[12] := FALSE;
   S701_RETURN_LOCK_ERR.Visu_Ret_Arr[13] := FALSE;
   S701_RETURN_LOCK_ERR.Visu_Ret_Arr[14] := FALSE;
   S701_RETURN_LOCK_ERR.Visu_Ret_Arr[15] := FALSE;
   S701_RETURN_LOCK_ERR.BLK_Move_Ret := 0;
   S701_RETURN_LOCK_ERR.Enable := FALSE;
   S701_RETURN_LOCK_ERR.Adv_End := FALSE;
   S701_RETURN_LOCK_ERR.Ret_End := FALSE;
   S701_TURN_LOCK_ERR.Enable_Aux := FALSE;
   S701_TURN_LOCK_ERR.Adv_Amount := 0;
   S701_TURN_LOCK_ERR.Ret_Amount := 0;
   S701_TURN_LOCK_ERR.LS_Adv1 := FALSE;
   S701_TURN_LOCK_ERR.LS_Ret1 := FALSE;
   S701_TURN_LOCK_ERR.LS_Adv2 := FALSE;
   S701_TURN_LOCK_ERR.LS_Ret2 := FALSE;
   S701_TURN_LOCK_ERR.LS_Adv3 := FALSE;
   S701_TURN_LOCK_ERR.LS_Ret3 := FALSE;
   S701_TURN_LOCK_ERR.LS_Adv4 := FALSE;
   S701_TURN_LOCK_ERR.LS_Ret4 := FALSE;
   S701_TURN_LOCK_ERR.SOL_Adv := FALSE;
   S701_TURN_LOCK_ERR.SOL_Ret := FALSE;
   S701_TURN_LOCK_ERR.M_Ready := FALSE;
   S701_TURN_LOCK_ERR.T_CHK1 := T#0MS;
   S701_TURN_LOCK_ERR.T_CHK2 := T#0MS;
   S701_TURN_LOCK_ERR.PB_Lamp_CHK := FALSE;
   S701_TURN_LOCK_ERR.PB_Error_Rst := FALSE;
   S701_TURN_LOCK_ERR.M_FLICK := FALSE;
   S701_TURN_LOCK_ERR.M_Adv_Err := FALSE;
   S701_TURN_LOCK_ERR.M_Ret_Err := FALSE;
   S701_TURN_LOCK_ERR.LP_Adv := FALSE;
   S701_TURN_LOCK_ERR.LP_Ret := FALSE;
   S701_TURN_LOCK_ERR.Visu_Adv := W#16#0;
   S701_TURN_LOCK_ERR.Visu_Ret := W#16#0;
   S701_TURN_LOCK_ERR.Error_T1.IN := FALSE;
   S701_TURN_LOCK_ERR.Error_T1.PT := T#0MS;
   S701_TURN_LOCK_ERR.Error_T1.Q := FALSE;
   S701_TURN_LOCK_ERR.Error_T1.ET := T#0MS;
   S701_TURN_LOCK_ERR.Error_T1.STATE := B#16#0;
   S701_TURN_LOCK_ERR.Error_T1.STIME := T#0MS;
   S701_TURN_LOCK_ERR.Error_T1.ATIME := T#0MS;
   S701_TURN_LOCK_ERR.Error_T2.IN := FALSE;
   S701_TURN_LOCK_ERR.Error_T2.PT := T#0MS;
   S701_TURN_LOCK_ERR.Error_T2.Q := FALSE;
   S701_TURN_LOCK_ERR.Error_T2.ET := T#0MS;
   S701_TURN_LOCK_ERR.Error_T2.STATE := B#16#0;
   S701_TURN_LOCK_ERR.Error_T2.STIME := T#0MS;
   S701_TURN_LOCK_ERR.Error_T2.ATIME := T#0MS;
   S701_TURN_LOCK_ERR.CHK_Aux1 := FALSE;
   S701_TURN_LOCK_ERR.CHK_Aux2 := FALSE;
   S701_TURN_LOCK_ERR.Error_T1_DN := FALSE;
   S701_TURN_LOCK_ERR.Error_T2_DN := FALSE;
   S701_TURN_LOCK_ERR.Adv_Memo := FALSE;
   S701_TURN_LOCK_ERR.Visu_Adv_Arr[0] := FALSE;
   S701_TURN_LOCK_ERR.Visu_Adv_Arr[1] := FALSE;
   S701_TURN_LOCK_ERR.Visu_Adv_Arr[2] := FALSE;
   S701_TURN_LOCK_ERR.Visu_Adv_Arr[3] := FALSE;
   S701_TURN_LOCK_ERR.Visu_Adv_Arr[4] := FALSE;
   S701_TURN_LOCK_ERR.Visu_Adv_Arr[5] := FALSE;
   S701_TURN_LOCK_ERR.Visu_Adv_Arr[6] := FALSE;
   S701_TURN_LOCK_ERR.Visu_Adv_Arr[7] := FALSE;
   S701_TURN_LOCK_ERR.Visu_Adv_Arr[8] := FALSE;
   S701_TURN_LOCK_ERR.Visu_Adv_Arr[9] := FALSE;
   S701_TURN_LOCK_ERR.Visu_Adv_Arr[10] := FALSE;
   S701_TURN_LOCK_ERR.Visu_Adv_Arr[11] := FALSE;
   S701_TURN_LOCK_ERR.Visu_Adv_Arr[12] := FALSE;
   S701_TURN_LOCK_ERR.Visu_Adv_Arr[13] := FALSE;
   S701_TURN_LOCK_ERR.Visu_Adv_Arr[14] := FALSE;
   S701_TURN_LOCK_ERR.Visu_Adv_Arr[15] := FALSE;
   S701_TURN_LOCK_ERR.Visu_Ret_Arr[0] := FALSE;
   S701_TURN_LOCK_ERR.Visu_Ret_Arr[1] := FALSE;
   S701_TURN_LOCK_ERR.Visu_Ret_Arr[2] := FALSE;
   S701_TURN_LOCK_ERR.Visu_Ret_Arr[3] := FALSE;
   S701_TURN_LOCK_ERR.Visu_Ret_Arr[4] := FALSE;
   S701_TURN_LOCK_ERR.Visu_Ret_Arr[5] := FALSE;
   S701_TURN_LOCK_ERR.Visu_Ret_Arr[6] := FALSE;
   S701_TURN_LOCK_ERR.Visu_Ret_Arr[7] := FALSE;
   S701_TURN_LOCK_ERR.Visu_Ret_Arr[8] := FALSE;
   S701_TURN_LOCK_ERR.Visu_Ret_Arr[9] := FALSE;
   S701_TURN_LOCK_ERR.Visu_Ret_Arr[10] := FALSE;
   S701_TURN_LOCK_ERR.Visu_Ret_Arr[11] := FALSE;
   S701_TURN_LOCK_ERR.Visu_Ret_Arr[12] := FALSE;
   S701_TURN_LOCK_ERR.Visu_Ret_Arr[13] := FALSE;
   S701_TURN_LOCK_ERR.Visu_Ret_Arr[14] := FALSE;
   S701_TURN_LOCK_ERR.Visu_Ret_Arr[15] := FALSE;
   S701_TURN_LOCK_ERR.BLK_Move_Ret := 0;
   S701_TURN_LOCK_ERR.Enable := FALSE;
   S701_TURN_LOCK_ERR.Adv_End := FALSE;
   S701_TURN_LOCK_ERR.Ret_End := FALSE;
   S701_LM_PIN1_ERR.Enable_Aux := FALSE;
   S701_LM_PIN1_ERR.Adv_Amount := 0;
   S701_LM_PIN1_ERR.Ret_Amount := 0;
   S701_LM_PIN1_ERR.LS_Adv1 := FALSE;
   S701_LM_PIN1_ERR.LS_Ret1 := FALSE;
   S701_LM_PIN1_ERR.LS_Adv2 := FALSE;
   S701_LM_PIN1_ERR.LS_Ret2 := FALSE;
   S701_LM_PIN1_ERR.LS_Adv3 := FALSE;
   S701_LM_PIN1_ERR.LS_Ret3 := FALSE;
   S701_LM_PIN1_ERR.LS_Adv4 := FALSE;
   S701_LM_PIN1_ERR.LS_Ret4 := FALSE;
   S701_LM_PIN1_ERR.SOL_Adv := FALSE;
   S701_LM_PIN1_ERR.SOL_Ret := FALSE;
   S701_LM_PIN1_ERR.M_Ready := FALSE;
   S701_LM_PIN1_ERR.T_CHK1 := T#0MS;
   S701_LM_PIN1_ERR.T_CHK2 := T#0MS;
   S701_LM_PIN1_ERR.PB_Lamp_CHK := FALSE;
   S701_LM_PIN1_ERR.PB_Error_Rst := FALSE;
   S701_LM_PIN1_ERR.M_FLICK := FALSE;
   S701_LM_PIN1_ERR.M_Adv_Err := FALSE;
   S701_LM_PIN1_ERR.M_Ret_Err := FALSE;
   S701_LM_PIN1_ERR.LP_Adv := FALSE;
   S701_LM_PIN1_ERR.LP_Ret := FALSE;
   S701_LM_PIN1_ERR.Visu_Adv := W#16#0;
   S701_LM_PIN1_ERR.Visu_Ret := W#16#0;
   S701_LM_PIN1_ERR.Error_T1.IN := FALSE;
   S701_LM_PIN1_ERR.Error_T1.PT := T#0MS;
   S701_LM_PIN1_ERR.Error_T1.Q := FALSE;
   S701_LM_PIN1_ERR.Error_T1.ET := T#0MS;
   S701_LM_PIN1_ERR.Error_T1.STATE := B#16#0;
   S701_LM_PIN1_ERR.Error_T1.STIME := T#0MS;
   S701_LM_PIN1_ERR.Error_T1.ATIME := T#0MS;
   S701_LM_PIN1_ERR.Error_T2.IN := FALSE;
   S701_LM_PIN1_ERR.Error_T2.PT := T#0MS;
   S701_LM_PIN1_ERR.Error_T2.Q := FALSE;
   S701_LM_PIN1_ERR.Error_T2.ET := T#0MS;
   S701_LM_PIN1_ERR.Error_T2.STATE := B#16#0;
   S701_LM_PIN1_ERR.Error_T2.STIME := T#0MS;
   S701_LM_PIN1_ERR.Error_T2.ATIME := T#0MS;
   S701_LM_PIN1_ERR.CHK_Aux1 := FALSE;
   S701_LM_PIN1_ERR.CHK_Aux2 := FALSE;
   S701_LM_PIN1_ERR.Error_T1_DN := FALSE;
   S701_LM_PIN1_ERR.Error_T2_DN := FALSE;
   S701_LM_PIN1_ERR.Adv_Memo := FALSE;
   S701_LM_PIN1_ERR.Visu_Adv_Arr[0] := FALSE;
   S701_LM_PIN1_ERR.Visu_Adv_Arr[1] := FALSE;
   S701_LM_PIN1_ERR.Visu_Adv_Arr[2] := FALSE;
   S701_LM_PIN1_ERR.Visu_Adv_Arr[3] := FALSE;
   S701_LM_PIN1_ERR.Visu_Adv_Arr[4] := FALSE;
   S701_LM_PIN1_ERR.Visu_Adv_Arr[5] := FALSE;
   S701_LM_PIN1_ERR.Visu_Adv_Arr[6] := FALSE;
   S701_LM_PIN1_ERR.Visu_Adv_Arr[7] := FALSE;
   S701_LM_PIN1_ERR.Visu_Adv_Arr[8] := FALSE;
   S701_LM_PIN1_ERR.Visu_Adv_Arr[9] := FALSE;
   S701_LM_PIN1_ERR.Visu_Adv_Arr[10] := FALSE;
   S701_LM_PIN1_ERR.Visu_Adv_Arr[11] := FALSE;
   S701_LM_PIN1_ERR.Visu_Adv_Arr[12] := FALSE;
   S701_LM_PIN1_ERR.Visu_Adv_Arr[13] := FALSE;
   S701_LM_PIN1_ERR.Visu_Adv_Arr[14] := FALSE;
   S701_LM_PIN1_ERR.Visu_Adv_Arr[15] := FALSE;
   S701_LM_PIN1_ERR.Visu_Ret_Arr[0] := FALSE;
   S701_LM_PIN1_ERR.Visu_Ret_Arr[1] := FALSE;
   S701_LM_PIN1_ERR.Visu_Ret_Arr[2] := FALSE;
   S701_LM_PIN1_ERR.Visu_Ret_Arr[3] := FALSE;
   S701_LM_PIN1_ERR.Visu_Ret_Arr[4] := FALSE;
   S701_LM_PIN1_ERR.Visu_Ret_Arr[5] := FALSE;
   S701_LM_PIN1_ERR.Visu_Ret_Arr[6] := FALSE;
   S701_LM_PIN1_ERR.Visu_Ret_Arr[7] := FALSE;
   S701_LM_PIN1_ERR.Visu_Ret_Arr[8] := FALSE;
   S701_LM_PIN1_ERR.Visu_Ret_Arr[9] := FALSE;
   S701_LM_PIN1_ERR.Visu_Ret_Arr[10] := FALSE;
   S701_LM_PIN1_ERR.Visu_Ret_Arr[11] := FALSE;
   S701_LM_PIN1_ERR.Visu_Ret_Arr[12] := FALSE;
   S701_LM_PIN1_ERR.Visu_Ret_Arr[13] := FALSE;
   S701_LM_PIN1_ERR.Visu_Ret_Arr[14] := FALSE;
   S701_LM_PIN1_ERR.Visu_Ret_Arr[15] := FALSE;
   S701_LM_PIN1_ERR.BLK_Move_Ret := 0;
   S701_LM_PIN1_ERR.Enable := FALSE;
   S701_LM_PIN1_ERR.Adv_End := FALSE;
   S701_LM_PIN1_ERR.Ret_End := FALSE;
   S701_LM_PIN2_ERR.Enable_Aux := FALSE;
   S701_LM_PIN2_ERR.Adv_Amount := 0;
   S701_LM_PIN2_ERR.Ret_Amount := 0;
   S701_LM_PIN2_ERR.LS_Adv1 := FALSE;
   S701_LM_PIN2_ERR.LS_Ret1 := FALSE;
   S701_LM_PIN2_ERR.LS_Adv2 := FALSE;
   S701_LM_PIN2_ERR.LS_Ret2 := FALSE;
   S701_LM_PIN2_ERR.LS_Adv3 := FALSE;
   S701_LM_PIN2_ERR.LS_Ret3 := FALSE;
   S701_LM_PIN2_ERR.LS_Adv4 := FALSE;
   S701_LM_PIN2_ERR.LS_Ret4 := FALSE;
   S701_LM_PIN2_ERR.SOL_Adv := FALSE;
   S701_LM_PIN2_ERR.SOL_Ret := FALSE;
   S701_LM_PIN2_ERR.M_Ready := FALSE;
   S701_LM_PIN2_ERR.T_CHK1 := T#0MS;
   S701_LM_PIN2_ERR.T_CHK2 := T#0MS;
   S701_LM_PIN2_ERR.PB_Lamp_CHK := FALSE;
   S701_LM_PIN2_ERR.PB_Error_Rst := FALSE;
   S701_LM_PIN2_ERR.M_FLICK := FALSE;
   S701_LM_PIN2_ERR.M_Adv_Err := FALSE;
   S701_LM_PIN2_ERR.M_Ret_Err := FALSE;
   S701_LM_PIN2_ERR.LP_Adv := FALSE;
   S701_LM_PIN2_ERR.LP_Ret := FALSE;
   S701_LM_PIN2_ERR.Visu_Adv := W#16#0;
   S701_LM_PIN2_ERR.Visu_Ret := W#16#0;
   S701_LM_PIN2_ERR.Error_T1.IN := FALSE;
   S701_LM_PIN2_ERR.Error_T1.PT := T#0MS;
   S701_LM_PIN2_ERR.Error_T1.Q := FALSE;
   S701_LM_PIN2_ERR.Error_T1.ET := T#0MS;
   S701_LM_PIN2_ERR.Error_T1.STATE := B#16#0;
   S701_LM_PIN2_ERR.Error_T1.STIME := T#0MS;
   S701_LM_PIN2_ERR.Error_T1.ATIME := T#0MS;
   S701_LM_PIN2_ERR.Error_T2.IN := FALSE;
   S701_LM_PIN2_ERR.Error_T2.PT := T#0MS;
   S701_LM_PIN2_ERR.Error_T2.Q := FALSE;
   S701_LM_PIN2_ERR.Error_T2.ET := T#0MS;
   S701_LM_PIN2_ERR.Error_T2.STATE := B#16#0;
   S701_LM_PIN2_ERR.Error_T2.STIME := T#0MS;
   S701_LM_PIN2_ERR.Error_T2.ATIME := T#0MS;
   S701_LM_PIN2_ERR.CHK_Aux1 := FALSE;
   S701_LM_PIN2_ERR.CHK_Aux2 := FALSE;
   S701_LM_PIN2_ERR.Error_T1_DN := FALSE;
   S701_LM_PIN2_ERR.Error_T2_DN := FALSE;
   S701_LM_PIN2_ERR.Adv_Memo := FALSE;
   S701_LM_PIN2_ERR.Visu_Adv_Arr[0] := FALSE;
   S701_LM_PIN2_ERR.Visu_Adv_Arr[1] := FALSE;
   S701_LM_PIN2_ERR.Visu_Adv_Arr[2] := FALSE;
   S701_LM_PIN2_ERR.Visu_Adv_Arr[3] := FALSE;
   S701_LM_PIN2_ERR.Visu_Adv_Arr[4] := FALSE;
   S701_LM_PIN2_ERR.Visu_Adv_Arr[5] := FALSE;
   S701_LM_PIN2_ERR.Visu_Adv_Arr[6] := FALSE;
   S701_LM_PIN2_ERR.Visu_Adv_Arr[7] := FALSE;
   S701_LM_PIN2_ERR.Visu_Adv_Arr[8] := FALSE;
   S701_LM_PIN2_ERR.Visu_Adv_Arr[9] := FALSE;
   S701_LM_PIN2_ERR.Visu_Adv_Arr[10] := FALSE;
   S701_LM_PIN2_ERR.Visu_Adv_Arr[11] := FALSE;
   S701_LM_PIN2_ERR.Visu_Adv_Arr[12] := FALSE;
   S701_LM_PIN2_ERR.Visu_Adv_Arr[13] := FALSE;
   S701_LM_PIN2_ERR.Visu_Adv_Arr[14] := FALSE;
   S701_LM_PIN2_ERR.Visu_Adv_Arr[15] := FALSE;
   S701_LM_PIN2_ERR.Visu_Ret_Arr[0] := FALSE;
   S701_LM_PIN2_ERR.Visu_Ret_Arr[1] := FALSE;
   S701_LM_PIN2_ERR.Visu_Ret_Arr[2] := FALSE;
   S701_LM_PIN2_ERR.Visu_Ret_Arr[3] := FALSE;
   S701_LM_PIN2_ERR.Visu_Ret_Arr[4] := FALSE;
   S701_LM_PIN2_ERR.Visu_Ret_Arr[5] := FALSE;
   S701_LM_PIN2_ERR.Visu_Ret_Arr[6] := FALSE;
   S701_LM_PIN2_ERR.Visu_Ret_Arr[7] := FALSE;
   S701_LM_PIN2_ERR.Visu_Ret_Arr[8] := FALSE;
   S701_LM_PIN2_ERR.Visu_Ret_Arr[9] := FALSE;
   S701_LM_PIN2_ERR.Visu_Ret_Arr[10] := FALSE;
   S701_LM_PIN2_ERR.Visu_Ret_Arr[11] := FALSE;
   S701_LM_PIN2_ERR.Visu_Ret_Arr[12] := FALSE;
   S701_LM_PIN2_ERR.Visu_Ret_Arr[13] := FALSE;
   S701_LM_PIN2_ERR.Visu_Ret_Arr[14] := FALSE;
   S701_LM_PIN2_ERR.Visu_Ret_Arr[15] := FALSE;
   S701_LM_PIN2_ERR.BLK_Move_Ret := 0;
   S701_LM_PIN2_ERR.Enable := FALSE;
   S701_LM_PIN2_ERR.Adv_End := FALSE;
   S701_LM_PIN2_ERR.Ret_End := FALSE;
   S701_LM_PIN3_ERR.Enable_Aux := FALSE;
   S701_LM_PIN3_ERR.Adv_Amount := 0;
   S701_LM_PIN3_ERR.Ret_Amount := 0;
   S701_LM_PIN3_ERR.LS_Adv1 := FALSE;
   S701_LM_PIN3_ERR.LS_Ret1 := FALSE;
   S701_LM_PIN3_ERR.LS_Adv2 := FALSE;
   S701_LM_PIN3_ERR.LS_Ret2 := FALSE;
   S701_LM_PIN3_ERR.LS_Adv3 := FALSE;
   S701_LM_PIN3_ERR.LS_Ret3 := FALSE;
   S701_LM_PIN3_ERR.LS_Adv4 := FALSE;
   S701_LM_PIN3_ERR.LS_Ret4 := FALSE;
   S701_LM_PIN3_ERR.SOL_Adv := FALSE;
   S701_LM_PIN3_ERR.SOL_Ret := FALSE;
   S701_LM_PIN3_ERR.M_Ready := FALSE;
   S701_LM_PIN3_ERR.T_CHK1 := T#0MS;
   S701_LM_PIN3_ERR.T_CHK2 := T#0MS;
   S701_LM_PIN3_ERR.PB_Lamp_CHK := FALSE;
   S701_LM_PIN3_ERR.PB_Error_Rst := FALSE;
   S701_LM_PIN3_ERR.M_FLICK := FALSE;
   S701_LM_PIN3_ERR.M_Adv_Err := FALSE;
   S701_LM_PIN3_ERR.M_Ret_Err := FALSE;
   S701_LM_PIN3_ERR.LP_Adv := FALSE;
   S701_LM_PIN3_ERR.LP_Ret := FALSE;
   S701_LM_PIN3_ERR.Visu_Adv := W#16#0;
   S701_LM_PIN3_ERR.Visu_Ret := W#16#0;
   S701_LM_PIN3_ERR.Error_T1.IN := FALSE;
   S701_LM_PIN3_ERR.Error_T1.PT := T#0MS;
   S701_LM_PIN3_ERR.Error_T1.Q := FALSE;
   S701_LM_PIN3_ERR.Error_T1.ET := T#0MS;
   S701_LM_PIN3_ERR.Error_T1.STATE := B#16#0;
   S701_LM_PIN3_ERR.Error_T1.STIME := T#0MS;
   S701_LM_PIN3_ERR.Error_T1.ATIME := T#0MS;
   S701_LM_PIN3_ERR.Error_T2.IN := FALSE;
   S701_LM_PIN3_ERR.Error_T2.PT := T#0MS;
   S701_LM_PIN3_ERR.Error_T2.Q := FALSE;
   S701_LM_PIN3_ERR.Error_T2.ET := T#0MS;
   S701_LM_PIN3_ERR.Error_T2.STATE := B#16#0;
   S701_LM_PIN3_ERR.Error_T2.STIME := T#0MS;
   S701_LM_PIN3_ERR.Error_T2.ATIME := T#0MS;
   S701_LM_PIN3_ERR.CHK_Aux1 := FALSE;
   S701_LM_PIN3_ERR.CHK_Aux2 := FALSE;
   S701_LM_PIN3_ERR.Error_T1_DN := FALSE;
   S701_LM_PIN3_ERR.Error_T2_DN := FALSE;
   S701_LM_PIN3_ERR.Adv_Memo := FALSE;
   S701_LM_PIN3_ERR.Visu_Adv_Arr[0] := FALSE;
   S701_LM_PIN3_ERR.Visu_Adv_Arr[1] := FALSE;
   S701_LM_PIN3_ERR.Visu_Adv_Arr[2] := FALSE;
   S701_LM_PIN3_ERR.Visu_Adv_Arr[3] := FALSE;
   S701_LM_PIN3_ERR.Visu_Adv_Arr[4] := FALSE;
   S701_LM_PIN3_ERR.Visu_Adv_Arr[5] := FALSE;
   S701_LM_PIN3_ERR.Visu_Adv_Arr[6] := FALSE;
   S701_LM_PIN3_ERR.Visu_Adv_Arr[7] := FALSE;
   S701_LM_PIN3_ERR.Visu_Adv_Arr[8] := FALSE;
   S701_LM_PIN3_ERR.Visu_Adv_Arr[9] := FALSE;
   S701_LM_PIN3_ERR.Visu_Adv_Arr[10] := FALSE;
   S701_LM_PIN3_ERR.Visu_Adv_Arr[11] := FALSE;
   S701_LM_PIN3_ERR.Visu_Adv_Arr[12] := FALSE;
   S701_LM_PIN3_ERR.Visu_Adv_Arr[13] := FALSE;
   S701_LM_PIN3_ERR.Visu_Adv_Arr[14] := FALSE;
   S701_LM_PIN3_ERR.Visu_Adv_Arr[15] := FALSE;
   S701_LM_PIN3_ERR.Visu_Ret_Arr[0] := FALSE;
   S701_LM_PIN3_ERR.Visu_Ret_Arr[1] := FALSE;
   S701_LM_PIN3_ERR.Visu_Ret_Arr[2] := FALSE;
   S701_LM_PIN3_ERR.Visu_Ret_Arr[3] := FALSE;
   S701_LM_PIN3_ERR.Visu_Ret_Arr[4] := FALSE;
   S701_LM_PIN3_ERR.Visu_Ret_Arr[5] := FALSE;
   S701_LM_PIN3_ERR.Visu_Ret_Arr[6] := FALSE;
   S701_LM_PIN3_ERR.Visu_Ret_Arr[7] := FALSE;
   S701_LM_PIN3_ERR.Visu_Ret_Arr[8] := FALSE;
   S701_LM_PIN3_ERR.Visu_Ret_Arr[9] := FALSE;
   S701_LM_PIN3_ERR.Visu_Ret_Arr[10] := FALSE;
   S701_LM_PIN3_ERR.Visu_Ret_Arr[11] := FALSE;
   S701_LM_PIN3_ERR.Visu_Ret_Arr[12] := FALSE;
   S701_LM_PIN3_ERR.Visu_Ret_Arr[13] := FALSE;
   S701_LM_PIN3_ERR.Visu_Ret_Arr[14] := FALSE;
   S701_LM_PIN3_ERR.Visu_Ret_Arr[15] := FALSE;
   S701_LM_PIN3_ERR.BLK_Move_Ret := 0;
   S701_LM_PIN3_ERR.Enable := FALSE;
   S701_LM_PIN3_ERR.Adv_End := FALSE;
   S701_LM_PIN3_ERR.Ret_End := FALSE;
   S701_LM_1_CLAMP1_ERR.Enable_Aux := FALSE;
   S701_LM_1_CLAMP1_ERR.Adv_Amount := 0;
   S701_LM_1_CLAMP1_ERR.Ret_Amount := 0;
   S701_LM_1_CLAMP1_ERR.LS_Adv1 := FALSE;
   S701_LM_1_CLAMP1_ERR.LS_Ret1 := FALSE;
   S701_LM_1_CLAMP1_ERR.LS_Adv2 := FALSE;
   S701_LM_1_CLAMP1_ERR.LS_Ret2 := FALSE;
   S701_LM_1_CLAMP1_ERR.LS_Adv3 := FALSE;
   S701_LM_1_CLAMP1_ERR.LS_Ret3 := FALSE;
   S701_LM_1_CLAMP1_ERR.LS_Adv4 := FALSE;
   S701_LM_1_CLAMP1_ERR.LS_Ret4 := FALSE;
   S701_LM_1_CLAMP1_ERR.SOL_Adv := FALSE;
   S701_LM_1_CLAMP1_ERR.SOL_Ret := FALSE;
   S701_LM_1_CLAMP1_ERR.M_Ready := FALSE;
   S701_LM_1_CLAMP1_ERR.T_CHK1 := T#0MS;
   S701_LM_1_CLAMP1_ERR.T_CHK2 := T#0MS;
   S701_LM_1_CLAMP1_ERR.PB_Lamp_CHK := FALSE;
   S701_LM_1_CLAMP1_ERR.PB_Error_Rst := FALSE;
   S701_LM_1_CLAMP1_ERR.M_FLICK := FALSE;
   S701_LM_1_CLAMP1_ERR.M_Adv_Err := FALSE;
   S701_LM_1_CLAMP1_ERR.M_Ret_Err := FALSE;
   S701_LM_1_CLAMP1_ERR.LP_Adv := FALSE;
   S701_LM_1_CLAMP1_ERR.LP_Ret := FALSE;
   S701_LM_1_CLAMP1_ERR.Visu_Adv := W#16#0;
   S701_LM_1_CLAMP1_ERR.Visu_Ret := W#16#0;
   S701_LM_1_CLAMP1_ERR.Error_T1.IN := FALSE;
   S701_LM_1_CLAMP1_ERR.Error_T1.PT := T#0MS;
   S701_LM_1_CLAMP1_ERR.Error_T1.Q := FALSE;
   S701_LM_1_CLAMP1_ERR.Error_T1.ET := T#0MS;
   S701_LM_1_CLAMP1_ERR.Error_T1.STATE := B#16#0;
   S701_LM_1_CLAMP1_ERR.Error_T1.STIME := T#0MS;
   S701_LM_1_CLAMP1_ERR.Error_T1.ATIME := T#0MS;
   S701_LM_1_CLAMP1_ERR.Error_T2.IN := FALSE;
   S701_LM_1_CLAMP1_ERR.Error_T2.PT := T#0MS;
   S701_LM_1_CLAMP1_ERR.Error_T2.Q := FALSE;
   S701_LM_1_CLAMP1_ERR.Error_T2.ET := T#0MS;
   S701_LM_1_CLAMP1_ERR.Error_T2.STATE := B#16#0;
   S701_LM_1_CLAMP1_ERR.Error_T2.STIME := T#0MS;
   S701_LM_1_CLAMP1_ERR.Error_T2.ATIME := T#0MS;
   S701_LM_1_CLAMP1_ERR.CHK_Aux1 := FALSE;
   S701_LM_1_CLAMP1_ERR.CHK_Aux2 := FALSE;
   S701_LM_1_CLAMP1_ERR.Error_T1_DN := FALSE;
   S701_LM_1_CLAMP1_ERR.Error_T2_DN := FALSE;
   S701_LM_1_CLAMP1_ERR.Adv_Memo := FALSE;
   S701_LM_1_CLAMP1_ERR.Visu_Adv_Arr[0] := FALSE;
   S701_LM_1_CLAMP1_ERR.Visu_Adv_Arr[1] := FALSE;
   S701_LM_1_CLAMP1_ERR.Visu_Adv_Arr[2] := FALSE;
   S701_LM_1_CLAMP1_ERR.Visu_Adv_Arr[3] := FALSE;
   S701_LM_1_CLAMP1_ERR.Visu_Adv_Arr[4] := FALSE;
   S701_LM_1_CLAMP1_ERR.Visu_Adv_Arr[5] := FALSE;
   S701_LM_1_CLAMP1_ERR.Visu_Adv_Arr[6] := FALSE;
   S701_LM_1_CLAMP1_ERR.Visu_Adv_Arr[7] := FALSE;
   S701_LM_1_CLAMP1_ERR.Visu_Adv_Arr[8] := FALSE;
   S701_LM_1_CLAMP1_ERR.Visu_Adv_Arr[9] := FALSE;
   S701_LM_1_CLAMP1_ERR.Visu_Adv_Arr[10] := FALSE;
   S701_LM_1_CLAMP1_ERR.Visu_Adv_Arr[11] := FALSE;
   S701_LM_1_CLAMP1_ERR.Visu_Adv_Arr[12] := FALSE;
   S701_LM_1_CLAMP1_ERR.Visu_Adv_Arr[13] := FALSE;
   S701_LM_1_CLAMP1_ERR.Visu_Adv_Arr[14] := FALSE;
   S701_LM_1_CLAMP1_ERR.Visu_Adv_Arr[15] := FALSE;
   S701_LM_1_CLAMP1_ERR.Visu_Ret_Arr[0] := FALSE;
   S701_LM_1_CLAMP1_ERR.Visu_Ret_Arr[1] := FALSE;
   S701_LM_1_CLAMP1_ERR.Visu_Ret_Arr[2] := FALSE;
   S701_LM_1_CLAMP1_ERR.Visu_Ret_Arr[3] := FALSE;
   S701_LM_1_CLAMP1_ERR.Visu_Ret_Arr[4] := FALSE;
   S701_LM_1_CLAMP1_ERR.Visu_Ret_Arr[5] := FALSE;
   S701_LM_1_CLAMP1_ERR.Visu_Ret_Arr[6] := FALSE;
   S701_LM_1_CLAMP1_ERR.Visu_Ret_Arr[7] := FALSE;
   S701_LM_1_CLAMP1_ERR.Visu_Ret_Arr[8] := FALSE;
   S701_LM_1_CLAMP1_ERR.Visu_Ret_Arr[9] := FALSE;
   S701_LM_1_CLAMP1_ERR.Visu_Ret_Arr[10] := FALSE;
   S701_LM_1_CLAMP1_ERR.Visu_Ret_Arr[11] := FALSE;
   S701_LM_1_CLAMP1_ERR.Visu_Ret_Arr[12] := FALSE;
   S701_LM_1_CLAMP1_ERR.Visu_Ret_Arr[13] := FALSE;
   S701_LM_1_CLAMP1_ERR.Visu_Ret_Arr[14] := FALSE;
   S701_LM_1_CLAMP1_ERR.Visu_Ret_Arr[15] := FALSE;
   S701_LM_1_CLAMP1_ERR.BLK_Move_Ret := 0;
   S701_LM_1_CLAMP1_ERR.Enable := FALSE;
   S701_LM_1_CLAMP1_ERR.Adv_End := FALSE;
   S701_LM_1_CLAMP1_ERR.Ret_End := FALSE;
   S701_LM_1_CLAMP2_ERR.Enable_Aux := FALSE;
   S701_LM_1_CLAMP2_ERR.Adv_Amount := 0;
   S701_LM_1_CLAMP2_ERR.Ret_Amount := 0;
   S701_LM_1_CLAMP2_ERR.LS_Adv1 := FALSE;
   S701_LM_1_CLAMP2_ERR.LS_Ret1 := FALSE;
   S701_LM_1_CLAMP2_ERR.LS_Adv2 := FALSE;
   S701_LM_1_CLAMP2_ERR.LS_Ret2 := FALSE;
   S701_LM_1_CLAMP2_ERR.LS_Adv3 := FALSE;
   S701_LM_1_CLAMP2_ERR.LS_Ret3 := FALSE;
   S701_LM_1_CLAMP2_ERR.LS_Adv4 := FALSE;
   S701_LM_1_CLAMP2_ERR.LS_Ret4 := FALSE;
   S701_LM_1_CLAMP2_ERR.SOL_Adv := FALSE;
   S701_LM_1_CLAMP2_ERR.SOL_Ret := FALSE;
   S701_LM_1_CLAMP2_ERR.M_Ready := FALSE;
   S701_LM_1_CLAMP2_ERR.T_CHK1 := T#0MS;
   S701_LM_1_CLAMP2_ERR.T_CHK2 := T#0MS;
   S701_LM_1_CLAMP2_ERR.PB_Lamp_CHK := FALSE;
   S701_LM_1_CLAMP2_ERR.PB_Error_Rst := FALSE;
   S701_LM_1_CLAMP2_ERR.M_FLICK := FALSE;
   S701_LM_1_CLAMP2_ERR.M_Adv_Err := FALSE;
   S701_LM_1_CLAMP2_ERR.M_Ret_Err := FALSE;
   S701_LM_1_CLAMP2_ERR.LP_Adv := FALSE;
   S701_LM_1_CLAMP2_ERR.LP_Ret := FALSE;
   S701_LM_1_CLAMP2_ERR.Visu_Adv := W#16#0;
   S701_LM_1_CLAMP2_ERR.Visu_Ret := W#16#0;
   S701_LM_1_CLAMP2_ERR.Error_T1.IN := FALSE;
   S701_LM_1_CLAMP2_ERR.Error_T1.PT := T#0MS;
   S701_LM_1_CLAMP2_ERR.Error_T1.Q := FALSE;
   S701_LM_1_CLAMP2_ERR.Error_T1.ET := T#0MS;
   S701_LM_1_CLAMP2_ERR.Error_T1.STATE := B#16#0;
   S701_LM_1_CLAMP2_ERR.Error_T1.STIME := T#0MS;
   S701_LM_1_CLAMP2_ERR.Error_T1.ATIME := T#0MS;
   S701_LM_1_CLAMP2_ERR.Error_T2.IN := FALSE;
   S701_LM_1_CLAMP2_ERR.Error_T2.PT := T#0MS;
   S701_LM_1_CLAMP2_ERR.Error_T2.Q := FALSE;
   S701_LM_1_CLAMP2_ERR.Error_T2.ET := T#0MS;
   S701_LM_1_CLAMP2_ERR.Error_T2.STATE := B#16#0;
   S701_LM_1_CLAMP2_ERR.Error_T2.STIME := T#0MS;
   S701_LM_1_CLAMP2_ERR.Error_T2.ATIME := T#0MS;
   S701_LM_1_CLAMP2_ERR.CHK_Aux1 := FALSE;
   S701_LM_1_CLAMP2_ERR.CHK_Aux2 := FALSE;
   S701_LM_1_CLAMP2_ERR.Error_T1_DN := FALSE;
   S701_LM_1_CLAMP2_ERR.Error_T2_DN := FALSE;
   S701_LM_1_CLAMP2_ERR.Adv_Memo := FALSE;
   S701_LM_1_CLAMP2_ERR.Visu_Adv_Arr[0] := FALSE;
   S701_LM_1_CLAMP2_ERR.Visu_Adv_Arr[1] := FALSE;
   S701_LM_1_CLAMP2_ERR.Visu_Adv_Arr[2] := FALSE;
   S701_LM_1_CLAMP2_ERR.Visu_Adv_Arr[3] := FALSE;
   S701_LM_1_CLAMP2_ERR.Visu_Adv_Arr[4] := FALSE;
   S701_LM_1_CLAMP2_ERR.Visu_Adv_Arr[5] := FALSE;
   S701_LM_1_CLAMP2_ERR.Visu_Adv_Arr[6] := FALSE;
   S701_LM_1_CLAMP2_ERR.Visu_Adv_Arr[7] := FALSE;
   S701_LM_1_CLAMP2_ERR.Visu_Adv_Arr[8] := FALSE;
   S701_LM_1_CLAMP2_ERR.Visu_Adv_Arr[9] := FALSE;
   S701_LM_1_CLAMP2_ERR.Visu_Adv_Arr[10] := FALSE;
   S701_LM_1_CLAMP2_ERR.Visu_Adv_Arr[11] := FALSE;
   S701_LM_1_CLAMP2_ERR.Visu_Adv_Arr[12] := FALSE;
   S701_LM_1_CLAMP2_ERR.Visu_Adv_Arr[13] := FALSE;
   S701_LM_1_CLAMP2_ERR.Visu_Adv_Arr[14] := FALSE;
   S701_LM_1_CLAMP2_ERR.Visu_Adv_Arr[15] := FALSE;
   S701_LM_1_CLAMP2_ERR.Visu_Ret_Arr[0] := FALSE;
   S701_LM_1_CLAMP2_ERR.Visu_Ret_Arr[1] := FALSE;
   S701_LM_1_CLAMP2_ERR.Visu_Ret_Arr[2] := FALSE;
   S701_LM_1_CLAMP2_ERR.Visu_Ret_Arr[3] := FALSE;
   S701_LM_1_CLAMP2_ERR.Visu_Ret_Arr[4] := FALSE;
   S701_LM_1_CLAMP2_ERR.Visu_Ret_Arr[5] := FALSE;
   S701_LM_1_CLAMP2_ERR.Visu_Ret_Arr[6] := FALSE;
   S701_LM_1_CLAMP2_ERR.Visu_Ret_Arr[7] := FALSE;
   S701_LM_1_CLAMP2_ERR.Visu_Ret_Arr[8] := FALSE;
   S701_LM_1_CLAMP2_ERR.Visu_Ret_Arr[9] := FALSE;
   S701_LM_1_CLAMP2_ERR.Visu_Ret_Arr[10] := FALSE;
   S701_LM_1_CLAMP2_ERR.Visu_Ret_Arr[11] := FALSE;
   S701_LM_1_CLAMP2_ERR.Visu_Ret_Arr[12] := FALSE;
   S701_LM_1_CLAMP2_ERR.Visu_Ret_Arr[13] := FALSE;
   S701_LM_1_CLAMP2_ERR.Visu_Ret_Arr[14] := FALSE;
   S701_LM_1_CLAMP2_ERR.Visu_Ret_Arr[15] := FALSE;
   S701_LM_1_CLAMP2_ERR.BLK_Move_Ret := 0;
   S701_LM_1_CLAMP2_ERR.Enable := FALSE;
   S701_LM_1_CLAMP2_ERR.Adv_End := FALSE;
   S701_LM_1_CLAMP2_ERR.Ret_End := FALSE;
   S701_LM_1_CLAMP3_ERR.Enable_Aux := FALSE;
   S701_LM_1_CLAMP3_ERR.Adv_Amount := 0;
   S701_LM_1_CLAMP3_ERR.Ret_Amount := 0;
   S701_LM_1_CLAMP3_ERR.LS_Adv1 := FALSE;
   S701_LM_1_CLAMP3_ERR.LS_Ret1 := FALSE;
   S701_LM_1_CLAMP3_ERR.LS_Adv2 := FALSE;
   S701_LM_1_CLAMP3_ERR.LS_Ret2 := FALSE;
   S701_LM_1_CLAMP3_ERR.LS_Adv3 := FALSE;
   S701_LM_1_CLAMP3_ERR.LS_Ret3 := FALSE;
   S701_LM_1_CLAMP3_ERR.LS_Adv4 := FALSE;
   S701_LM_1_CLAMP3_ERR.LS_Ret4 := FALSE;
   S701_LM_1_CLAMP3_ERR.SOL_Adv := FALSE;
   S701_LM_1_CLAMP3_ERR.SOL_Ret := FALSE;
   S701_LM_1_CLAMP3_ERR.M_Ready := FALSE;
   S701_LM_1_CLAMP3_ERR.T_CHK1 := T#0MS;
   S701_LM_1_CLAMP3_ERR.T_CHK2 := T#0MS;
   S701_LM_1_CLAMP3_ERR.PB_Lamp_CHK := FALSE;
   S701_LM_1_CLAMP3_ERR.PB_Error_Rst := FALSE;
   S701_LM_1_CLAMP3_ERR.M_FLICK := FALSE;
   S701_LM_1_CLAMP3_ERR.M_Adv_Err := FALSE;
   S701_LM_1_CLAMP3_ERR.M_Ret_Err := FALSE;
   S701_LM_1_CLAMP3_ERR.LP_Adv := FALSE;
   S701_LM_1_CLAMP3_ERR.LP_Ret := FALSE;
   S701_LM_1_CLAMP3_ERR.Visu_Adv := W#16#0;
   S701_LM_1_CLAMP3_ERR.Visu_Ret := W#16#0;
   S701_LM_1_CLAMP3_ERR.Error_T1.IN := FALSE;
   S701_LM_1_CLAMP3_ERR.Error_T1.PT := T#0MS;
   S701_LM_1_CLAMP3_ERR.Error_T1.Q := FALSE;
   S701_LM_1_CLAMP3_ERR.Error_T1.ET := T#0MS;
   S701_LM_1_CLAMP3_ERR.Error_T1.STATE := B#16#0;
   S701_LM_1_CLAMP3_ERR.Error_T1.STIME := T#0MS;
   S701_LM_1_CLAMP3_ERR.Error_T1.ATIME := T#0MS;
   S701_LM_1_CLAMP3_ERR.Error_T2.IN := FALSE;
   S701_LM_1_CLAMP3_ERR.Error_T2.PT := T#0MS;
   S701_LM_1_CLAMP3_ERR.Error_T2.Q := FALSE;
   S701_LM_1_CLAMP3_ERR.Error_T2.ET := T#0MS;
   S701_LM_1_CLAMP3_ERR.Error_T2.STATE := B#16#0;
   S701_LM_1_CLAMP3_ERR.Error_T2.STIME := T#0MS;
   S701_LM_1_CLAMP3_ERR.Error_T2.ATIME := T#0MS;
   S701_LM_1_CLAMP3_ERR.CHK_Aux1 := FALSE;
   S701_LM_1_CLAMP3_ERR.CHK_Aux2 := FALSE;
   S701_LM_1_CLAMP3_ERR.Error_T1_DN := FALSE;
   S701_LM_1_CLAMP3_ERR.Error_T2_DN := FALSE;
   S701_LM_1_CLAMP3_ERR.Adv_Memo := FALSE;
   S701_LM_1_CLAMP3_ERR.Visu_Adv_Arr[0] := FALSE;
   S701_LM_1_CLAMP3_ERR.Visu_Adv_Arr[1] := FALSE;
   S701_LM_1_CLAMP3_ERR.Visu_Adv_Arr[2] := FALSE;
   S701_LM_1_CLAMP3_ERR.Visu_Adv_Arr[3] := FALSE;
   S701_LM_1_CLAMP3_ERR.Visu_Adv_Arr[4] := FALSE;
   S701_LM_1_CLAMP3_ERR.Visu_Adv_Arr[5] := FALSE;
   S701_LM_1_CLAMP3_ERR.Visu_Adv_Arr[6] := FALSE;
   S701_LM_1_CLAMP3_ERR.Visu_Adv_Arr[7] := FALSE;
   S701_LM_1_CLAMP3_ERR.Visu_Adv_Arr[8] := FALSE;
   S701_LM_1_CLAMP3_ERR.Visu_Adv_Arr[9] := FALSE;
   S701_LM_1_CLAMP3_ERR.Visu_Adv_Arr[10] := FALSE;
   S701_LM_1_CLAMP3_ERR.Visu_Adv_Arr[11] := FALSE;
   S701_LM_1_CLAMP3_ERR.Visu_Adv_Arr[12] := FALSE;
   S701_LM_1_CLAMP3_ERR.Visu_Adv_Arr[13] := FALSE;
   S701_LM_1_CLAMP3_ERR.Visu_Adv_Arr[14] := FALSE;
   S701_LM_1_CLAMP3_ERR.Visu_Adv_Arr[15] := FALSE;
   S701_LM_1_CLAMP3_ERR.Visu_Ret_Arr[0] := FALSE;
   S701_LM_1_CLAMP3_ERR.Visu_Ret_Arr[1] := FALSE;
   S701_LM_1_CLAMP3_ERR.Visu_Ret_Arr[2] := FALSE;
   S701_LM_1_CLAMP3_ERR.Visu_Ret_Arr[3] := FALSE;
   S701_LM_1_CLAMP3_ERR.Visu_Ret_Arr[4] := FALSE;
   S701_LM_1_CLAMP3_ERR.Visu_Ret_Arr[5] := FALSE;
   S701_LM_1_CLAMP3_ERR.Visu_Ret_Arr[6] := FALSE;
   S701_LM_1_CLAMP3_ERR.Visu_Ret_Arr[7] := FALSE;
   S701_LM_1_CLAMP3_ERR.Visu_Ret_Arr[8] := FALSE;
   S701_LM_1_CLAMP3_ERR.Visu_Ret_Arr[9] := FALSE;
   S701_LM_1_CLAMP3_ERR.Visu_Ret_Arr[10] := FALSE;
   S701_LM_1_CLAMP3_ERR.Visu_Ret_Arr[11] := FALSE;
   S701_LM_1_CLAMP3_ERR.Visu_Ret_Arr[12] := FALSE;
   S701_LM_1_CLAMP3_ERR.Visu_Ret_Arr[13] := FALSE;
   S701_LM_1_CLAMP3_ERR.Visu_Ret_Arr[14] := FALSE;
   S701_LM_1_CLAMP3_ERR.Visu_Ret_Arr[15] := FALSE;
   S701_LM_1_CLAMP3_ERR.BLK_Move_Ret := 0;
   S701_LM_1_CLAMP3_ERR.Enable := FALSE;
   S701_LM_1_CLAMP3_ERR.Adv_End := FALSE;
   S701_LM_1_CLAMP3_ERR.Ret_End := FALSE;
   S701_LM_1_CLAMP4_ERR.Enable_Aux := FALSE;
   S701_LM_1_CLAMP4_ERR.Adv_Amount := 0;
   S701_LM_1_CLAMP4_ERR.Ret_Amount := 0;
   S701_LM_1_CLAMP4_ERR.LS_Adv1 := FALSE;
   S701_LM_1_CLAMP4_ERR.LS_Ret1 := FALSE;
   S701_LM_1_CLAMP4_ERR.LS_Adv2 := FALSE;
   S701_LM_1_CLAMP4_ERR.LS_Ret2 := FALSE;
   S701_LM_1_CLAMP4_ERR.LS_Adv3 := FALSE;
   S701_LM_1_CLAMP4_ERR.LS_Ret3 := FALSE;
   S701_LM_1_CLAMP4_ERR.LS_Adv4 := FALSE;
   S701_LM_1_CLAMP4_ERR.LS_Ret4 := FALSE;
   S701_LM_1_CLAMP4_ERR.SOL_Adv := FALSE;
   S701_LM_1_CLAMP4_ERR.SOL_Ret := FALSE;
   S701_LM_1_CLAMP4_ERR.M_Ready := FALSE;
   S701_LM_1_CLAMP4_ERR.T_CHK1 := T#0MS;
   S701_LM_1_CLAMP4_ERR.T_CHK2 := T#0MS;
   S701_LM_1_CLAMP4_ERR.PB_Lamp_CHK := FALSE;
   S701_LM_1_CLAMP4_ERR.PB_Error_Rst := FALSE;
   S701_LM_1_CLAMP4_ERR.M_FLICK := FALSE;
   S701_LM_1_CLAMP4_ERR.M_Adv_Err := FALSE;
   S701_LM_1_CLAMP4_ERR.M_Ret_Err := FALSE;
   S701_LM_1_CLAMP4_ERR.LP_Adv := FALSE;
   S701_LM_1_CLAMP4_ERR.LP_Ret := FALSE;
   S701_LM_1_CLAMP4_ERR.Visu_Adv := W#16#0;
   S701_LM_1_CLAMP4_ERR.Visu_Ret := W#16#0;
   S701_LM_1_CLAMP4_ERR.Error_T1.IN := FALSE;
   S701_LM_1_CLAMP4_ERR.Error_T1.PT := T#0MS;
   S701_LM_1_CLAMP4_ERR.Error_T1.Q := FALSE;
   S701_LM_1_CLAMP4_ERR.Error_T1.ET := T#0MS;
   S701_LM_1_CLAMP4_ERR.Error_T1.STATE := B#16#0;
   S701_LM_1_CLAMP4_ERR.Error_T1.STIME := T#0MS;
   S701_LM_1_CLAMP4_ERR.Error_T1.ATIME := T#0MS;
   S701_LM_1_CLAMP4_ERR.Error_T2.IN := FALSE;
   S701_LM_1_CLAMP4_ERR.Error_T2.PT := T#0MS;
   S701_LM_1_CLAMP4_ERR.Error_T2.Q := FALSE;
   S701_LM_1_CLAMP4_ERR.Error_T2.ET := T#0MS;
   S701_LM_1_CLAMP4_ERR.Error_T2.STATE := B#16#0;
   S701_LM_1_CLAMP4_ERR.Error_T2.STIME := T#0MS;
   S701_LM_1_CLAMP4_ERR.Error_T2.ATIME := T#0MS;
   S701_LM_1_CLAMP4_ERR.CHK_Aux1 := FALSE;
   S701_LM_1_CLAMP4_ERR.CHK_Aux2 := FALSE;
   S701_LM_1_CLAMP4_ERR.Error_T1_DN := FALSE;
   S701_LM_1_CLAMP4_ERR.Error_T2_DN := FALSE;
   S701_LM_1_CLAMP4_ERR.Adv_Memo := FALSE;
   S701_LM_1_CLAMP4_ERR.Visu_Adv_Arr[0] := FALSE;
   S701_LM_1_CLAMP4_ERR.Visu_Adv_Arr[1] := FALSE;
   S701_LM_1_CLAMP4_ERR.Visu_Adv_Arr[2] := FALSE;
   S701_LM_1_CLAMP4_ERR.Visu_Adv_Arr[3] := FALSE;
   S701_LM_1_CLAMP4_ERR.Visu_Adv_Arr[4] := FALSE;
   S701_LM_1_CLAMP4_ERR.Visu_Adv_Arr[5] := FALSE;
   S701_LM_1_CLAMP4_ERR.Visu_Adv_Arr[6] := FALSE;
   S701_LM_1_CLAMP4_ERR.Visu_Adv_Arr[7] := FALSE;
   S701_LM_1_CLAMP4_ERR.Visu_Adv_Arr[8] := FALSE;
   S701_LM_1_CLAMP4_ERR.Visu_Adv_Arr[9] := FALSE;
   S701_LM_1_CLAMP4_ERR.Visu_Adv_Arr[10] := FALSE;
   S701_LM_1_CLAMP4_ERR.Visu_Adv_Arr[11] := FALSE;
   S701_LM_1_CLAMP4_ERR.Visu_Adv_Arr[12] := FALSE;
   S701_LM_1_CLAMP4_ERR.Visu_Adv_Arr[13] := FALSE;
   S701_LM_1_CLAMP4_ERR.Visu_Adv_Arr[14] := FALSE;
   S701_LM_1_CLAMP4_ERR.Visu_Adv_Arr[15] := FALSE;
   S701_LM_1_CLAMP4_ERR.Visu_Ret_Arr[0] := FALSE;
   S701_LM_1_CLAMP4_ERR.Visu_Ret_Arr[1] := FALSE;
   S701_LM_1_CLAMP4_ERR.Visu_Ret_Arr[2] := FALSE;
   S701_LM_1_CLAMP4_ERR.Visu_Ret_Arr[3] := FALSE;
   S701_LM_1_CLAMP4_ERR.Visu_Ret_Arr[4] := FALSE;
   S701_LM_1_CLAMP4_ERR.Visu_Ret_Arr[5] := FALSE;
   S701_LM_1_CLAMP4_ERR.Visu_Ret_Arr[6] := FALSE;
   S701_LM_1_CLAMP4_ERR.Visu_Ret_Arr[7] := FALSE;
   S701_LM_1_CLAMP4_ERR.Visu_Ret_Arr[8] := FALSE;
   S701_LM_1_CLAMP4_ERR.Visu_Ret_Arr[9] := FALSE;
   S701_LM_1_CLAMP4_ERR.Visu_Ret_Arr[10] := FALSE;
   S701_LM_1_CLAMP4_ERR.Visu_Ret_Arr[11] := FALSE;
   S701_LM_1_CLAMP4_ERR.Visu_Ret_Arr[12] := FALSE;
   S701_LM_1_CLAMP4_ERR.Visu_Ret_Arr[13] := FALSE;
   S701_LM_1_CLAMP4_ERR.Visu_Ret_Arr[14] := FALSE;
   S701_LM_1_CLAMP4_ERR.Visu_Ret_Arr[15] := FALSE;
   S701_LM_1_CLAMP4_ERR.BLK_Move_Ret := 0;
   S701_LM_1_CLAMP4_ERR.Enable := FALSE;
   S701_LM_1_CLAMP4_ERR.Adv_End := FALSE;
   S701_LM_1_CLAMP4_ERR.Ret_End := FALSE;
   S701_LM_2_CLAMP1_ERR.Enable_Aux := FALSE;
   S701_LM_2_CLAMP1_ERR.Adv_Amount := 0;
   S701_LM_2_CLAMP1_ERR.Ret_Amount := 0;
   S701_LM_2_CLAMP1_ERR.LS_Adv1 := FALSE;
   S701_LM_2_CLAMP1_ERR.LS_Ret1 := FALSE;
   S701_LM_2_CLAMP1_ERR.LS_Adv2 := FALSE;
   S701_LM_2_CLAMP1_ERR.LS_Ret2 := FALSE;
   S701_LM_2_CLAMP1_ERR.LS_Adv3 := FALSE;
   S701_LM_2_CLAMP1_ERR.LS_Ret3 := FALSE;
   S701_LM_2_CLAMP1_ERR.LS_Adv4 := FALSE;
   S701_LM_2_CLAMP1_ERR.LS_Ret4 := FALSE;
   S701_LM_2_CLAMP1_ERR.SOL_Adv := FALSE;
   S701_LM_2_CLAMP1_ERR.SOL_Ret := FALSE;
   S701_LM_2_CLAMP1_ERR.M_Ready := FALSE;
   S701_LM_2_CLAMP1_ERR.T_CHK1 := T#0MS;
   S701_LM_2_CLAMP1_ERR.T_CHK2 := T#0MS;
   S701_LM_2_CLAMP1_ERR.PB_Lamp_CHK := FALSE;
   S701_LM_2_CLAMP1_ERR.PB_Error_Rst := FALSE;
   S701_LM_2_CLAMP1_ERR.M_FLICK := FALSE;
   S701_LM_2_CLAMP1_ERR.M_Adv_Err := FALSE;
   S701_LM_2_CLAMP1_ERR.M_Ret_Err := FALSE;
   S701_LM_2_CLAMP1_ERR.LP_Adv := FALSE;
   S701_LM_2_CLAMP1_ERR.LP_Ret := FALSE;
   S701_LM_2_CLAMP1_ERR.Visu_Adv := W#16#0;
   S701_LM_2_CLAMP1_ERR.Visu_Ret := W#16#0;
   S701_LM_2_CLAMP1_ERR.Error_T1.IN := FALSE;
   S701_LM_2_CLAMP1_ERR.Error_T1.PT := T#0MS;
   S701_LM_2_CLAMP1_ERR.Error_T1.Q := FALSE;
   S701_LM_2_CLAMP1_ERR.Error_T1.ET := T#0MS;
   S701_LM_2_CLAMP1_ERR.Error_T1.STATE := B#16#0;
   S701_LM_2_CLAMP1_ERR.Error_T1.STIME := T#0MS;
   S701_LM_2_CLAMP1_ERR.Error_T1.ATIME := T#0MS;
   S701_LM_2_CLAMP1_ERR.Error_T2.IN := FALSE;
   S701_LM_2_CLAMP1_ERR.Error_T2.PT := T#0MS;
   S701_LM_2_CLAMP1_ERR.Error_T2.Q := FALSE;
   S701_LM_2_CLAMP1_ERR.Error_T2.ET := T#0MS;
   S701_LM_2_CLAMP1_ERR.Error_T2.STATE := B#16#0;
   S701_LM_2_CLAMP1_ERR.Error_T2.STIME := T#0MS;
   S701_LM_2_CLAMP1_ERR.Error_T2.ATIME := T#0MS;
   S701_LM_2_CLAMP1_ERR.CHK_Aux1 := FALSE;
   S701_LM_2_CLAMP1_ERR.CHK_Aux2 := FALSE;
   S701_LM_2_CLAMP1_ERR.Error_T1_DN := FALSE;
   S701_LM_2_CLAMP1_ERR.Error_T2_DN := FALSE;
   S701_LM_2_CLAMP1_ERR.Adv_Memo := FALSE;
   S701_LM_2_CLAMP1_ERR.Visu_Adv_Arr[0] := FALSE;
   S701_LM_2_CLAMP1_ERR.Visu_Adv_Arr[1] := FALSE;
   S701_LM_2_CLAMP1_ERR.Visu_Adv_Arr[2] := FALSE;
   S701_LM_2_CLAMP1_ERR.Visu_Adv_Arr[3] := FALSE;
   S701_LM_2_CLAMP1_ERR.Visu_Adv_Arr[4] := FALSE;
   S701_LM_2_CLAMP1_ERR.Visu_Adv_Arr[5] := FALSE;
   S701_LM_2_CLAMP1_ERR.Visu_Adv_Arr[6] := FALSE;
   S701_LM_2_CLAMP1_ERR.Visu_Adv_Arr[7] := FALSE;
   S701_LM_2_CLAMP1_ERR.Visu_Adv_Arr[8] := FALSE;
   S701_LM_2_CLAMP1_ERR.Visu_Adv_Arr[9] := FALSE;
   S701_LM_2_CLAMP1_ERR.Visu_Adv_Arr[10] := FALSE;
   S701_LM_2_CLAMP1_ERR.Visu_Adv_Arr[11] := FALSE;
   S701_LM_2_CLAMP1_ERR.Visu_Adv_Arr[12] := FALSE;
   S701_LM_2_CLAMP1_ERR.Visu_Adv_Arr[13] := FALSE;
   S701_LM_2_CLAMP1_ERR.Visu_Adv_Arr[14] := FALSE;
   S701_LM_2_CLAMP1_ERR.Visu_Adv_Arr[15] := FALSE;
   S701_LM_2_CLAMP1_ERR.Visu_Ret_Arr[0] := FALSE;
   S701_LM_2_CLAMP1_ERR.Visu_Ret_Arr[1] := FALSE;
   S701_LM_2_CLAMP1_ERR.Visu_Ret_Arr[2] := FALSE;
   S701_LM_2_CLAMP1_ERR.Visu_Ret_Arr[3] := FALSE;
   S701_LM_2_CLAMP1_ERR.Visu_Ret_Arr[4] := FALSE;
   S701_LM_2_CLAMP1_ERR.Visu_Ret_Arr[5] := FALSE;
   S701_LM_2_CLAMP1_ERR.Visu_Ret_Arr[6] := FALSE;
   S701_LM_2_CLAMP1_ERR.Visu_Ret_Arr[7] := FALSE;
   S701_LM_2_CLAMP1_ERR.Visu_Ret_Arr[8] := FALSE;
   S701_LM_2_CLAMP1_ERR.Visu_Ret_Arr[9] := FALSE;
   S701_LM_2_CLAMP1_ERR.Visu_Ret_Arr[10] := FALSE;
   S701_LM_2_CLAMP1_ERR.Visu_Ret_Arr[11] := FALSE;
   S701_LM_2_CLAMP1_ERR.Visu_Ret_Arr[12] := FALSE;
   S701_LM_2_CLAMP1_ERR.Visu_Ret_Arr[13] := FALSE;
   S701_LM_2_CLAMP1_ERR.Visu_Ret_Arr[14] := FALSE;
   S701_LM_2_CLAMP1_ERR.Visu_Ret_Arr[15] := FALSE;
   S701_LM_2_CLAMP1_ERR.BLK_Move_Ret := 0;
   S701_LM_2_CLAMP1_ERR.Enable := FALSE;
   S701_LM_2_CLAMP1_ERR.Adv_End := FALSE;
   S701_LM_2_CLAMP1_ERR.Ret_End := FALSE;
   S701_LM_2_CLAMP2_ERR.Enable_Aux := FALSE;
   S701_LM_2_CLAMP2_ERR.Adv_Amount := 0;
   S701_LM_2_CLAMP2_ERR.Ret_Amount := 0;
   S701_LM_2_CLAMP2_ERR.LS_Adv1 := FALSE;
   S701_LM_2_CLAMP2_ERR.LS_Ret1 := FALSE;
   S701_LM_2_CLAMP2_ERR.LS_Adv2 := FALSE;
   S701_LM_2_CLAMP2_ERR.LS_Ret2 := FALSE;
   S701_LM_2_CLAMP2_ERR.LS_Adv3 := FALSE;
   S701_LM_2_CLAMP2_ERR.LS_Ret3 := FALSE;
   S701_LM_2_CLAMP2_ERR.LS_Adv4 := FALSE;
   S701_LM_2_CLAMP2_ERR.LS_Ret4 := FALSE;
   S701_LM_2_CLAMP2_ERR.SOL_Adv := FALSE;
   S701_LM_2_CLAMP2_ERR.SOL_Ret := FALSE;
   S701_LM_2_CLAMP2_ERR.M_Ready := FALSE;
   S701_LM_2_CLAMP2_ERR.T_CHK1 := T#0MS;
   S701_LM_2_CLAMP2_ERR.T_CHK2 := T#0MS;
   S701_LM_2_CLAMP2_ERR.PB_Lamp_CHK := FALSE;
   S701_LM_2_CLAMP2_ERR.PB_Error_Rst := FALSE;
   S701_LM_2_CLAMP2_ERR.M_FLICK := FALSE;
   S701_LM_2_CLAMP2_ERR.M_Adv_Err := FALSE;
   S701_LM_2_CLAMP2_ERR.M_Ret_Err := FALSE;
   S701_LM_2_CLAMP2_ERR.LP_Adv := FALSE;
   S701_LM_2_CLAMP2_ERR.LP_Ret := FALSE;
   S701_LM_2_CLAMP2_ERR.Visu_Adv := W#16#0;
   S701_LM_2_CLAMP2_ERR.Visu_Ret := W#16#0;
   S701_LM_2_CLAMP2_ERR.Error_T1.IN := FALSE;
   S701_LM_2_CLAMP2_ERR.Error_T1.PT := T#0MS;
   S701_LM_2_CLAMP2_ERR.Error_T1.Q := FALSE;
   S701_LM_2_CLAMP2_ERR.Error_T1.ET := T#0MS;
   S701_LM_2_CLAMP2_ERR.Error_T1.STATE := B#16#0;
   S701_LM_2_CLAMP2_ERR.Error_T1.STIME := T#0MS;
   S701_LM_2_CLAMP2_ERR.Error_T1.ATIME := T#0MS;
   S701_LM_2_CLAMP2_ERR.Error_T2.IN := FALSE;
   S701_LM_2_CLAMP2_ERR.Error_T2.PT := T#0MS;
   S701_LM_2_CLAMP2_ERR.Error_T2.Q := FALSE;
   S701_LM_2_CLAMP2_ERR.Error_T2.ET := T#0MS;
   S701_LM_2_CLAMP2_ERR.Error_T2.STATE := B#16#0;
   S701_LM_2_CLAMP2_ERR.Error_T2.STIME := T#0MS;
   S701_LM_2_CLAMP2_ERR.Error_T2.ATIME := T#0MS;
   S701_LM_2_CLAMP2_ERR.CHK_Aux1 := FALSE;
   S701_LM_2_CLAMP2_ERR.CHK_Aux2 := FALSE;
   S701_LM_2_CLAMP2_ERR.Error_T1_DN := FALSE;
   S701_LM_2_CLAMP2_ERR.Error_T2_DN := FALSE;
   S701_LM_2_CLAMP2_ERR.Adv_Memo := FALSE;
   S701_LM_2_CLAMP2_ERR.Visu_Adv_Arr[0] := FALSE;
   S701_LM_2_CLAMP2_ERR.Visu_Adv_Arr[1] := FALSE;
   S701_LM_2_CLAMP2_ERR.Visu_Adv_Arr[2] := FALSE;
   S701_LM_2_CLAMP2_ERR.Visu_Adv_Arr[3] := FALSE;
   S701_LM_2_CLAMP2_ERR.Visu_Adv_Arr[4] := FALSE;
   S701_LM_2_CLAMP2_ERR.Visu_Adv_Arr[5] := FALSE;
   S701_LM_2_CLAMP2_ERR.Visu_Adv_Arr[6] := FALSE;
   S701_LM_2_CLAMP2_ERR.Visu_Adv_Arr[7] := FALSE;
   S701_LM_2_CLAMP2_ERR.Visu_Adv_Arr[8] := FALSE;
   S701_LM_2_CLAMP2_ERR.Visu_Adv_Arr[9] := FALSE;
   S701_LM_2_CLAMP2_ERR.Visu_Adv_Arr[10] := FALSE;
   S701_LM_2_CLAMP2_ERR.Visu_Adv_Arr[11] := FALSE;
   S701_LM_2_CLAMP2_ERR.Visu_Adv_Arr[12] := FALSE;
   S701_LM_2_CLAMP2_ERR.Visu_Adv_Arr[13] := FALSE;
   S701_LM_2_CLAMP2_ERR.Visu_Adv_Arr[14] := FALSE;
   S701_LM_2_CLAMP2_ERR.Visu_Adv_Arr[15] := FALSE;
   S701_LM_2_CLAMP2_ERR.Visu_Ret_Arr[0] := FALSE;
   S701_LM_2_CLAMP2_ERR.Visu_Ret_Arr[1] := FALSE;
   S701_LM_2_CLAMP2_ERR.Visu_Ret_Arr[2] := FALSE;
   S701_LM_2_CLAMP2_ERR.Visu_Ret_Arr[3] := FALSE;
   S701_LM_2_CLAMP2_ERR.Visu_Ret_Arr[4] := FALSE;
   S701_LM_2_CLAMP2_ERR.Visu_Ret_Arr[5] := FALSE;
   S701_LM_2_CLAMP2_ERR.Visu_Ret_Arr[6] := FALSE;
   S701_LM_2_CLAMP2_ERR.Visu_Ret_Arr[7] := FALSE;
   S701_LM_2_CLAMP2_ERR.Visu_Ret_Arr[8] := FALSE;
   S701_LM_2_CLAMP2_ERR.Visu_Ret_Arr[9] := FALSE;
   S701_LM_2_CLAMP2_ERR.Visu_Ret_Arr[10] := FALSE;
   S701_LM_2_CLAMP2_ERR.Visu_Ret_Arr[11] := FALSE;
   S701_LM_2_CLAMP2_ERR.Visu_Ret_Arr[12] := FALSE;
   S701_LM_2_CLAMP2_ERR.Visu_Ret_Arr[13] := FALSE;
   S701_LM_2_CLAMP2_ERR.Visu_Ret_Arr[14] := FALSE;
   S701_LM_2_CLAMP2_ERR.Visu_Ret_Arr[15] := FALSE;
   S701_LM_2_CLAMP2_ERR.BLK_Move_Ret := 0;
   S701_LM_2_CLAMP2_ERR.Enable := FALSE;
   S701_LM_2_CLAMP2_ERR.Adv_End := FALSE;
   S701_LM_2_CLAMP2_ERR.Ret_End := FALSE;
   S701_LM_2_CLAMP3_ERR.Enable_Aux := FALSE;
   S701_LM_2_CLAMP3_ERR.Adv_Amount := 0;
   S701_LM_2_CLAMP3_ERR.Ret_Amount := 0;
   S701_LM_2_CLAMP3_ERR.LS_Adv1 := FALSE;
   S701_LM_2_CLAMP3_ERR.LS_Ret1 := FALSE;
   S701_LM_2_CLAMP3_ERR.LS_Adv2 := FALSE;
   S701_LM_2_CLAMP3_ERR.LS_Ret2 := FALSE;
   S701_LM_2_CLAMP3_ERR.LS_Adv3 := FALSE;
   S701_LM_2_CLAMP3_ERR.LS_Ret3 := FALSE;
   S701_LM_2_CLAMP3_ERR.LS_Adv4 := FALSE;
   S701_LM_2_CLAMP3_ERR.LS_Ret4 := FALSE;
   S701_LM_2_CLAMP3_ERR.SOL_Adv := FALSE;
   S701_LM_2_CLAMP3_ERR.SOL_Ret := FALSE;
   S701_LM_2_CLAMP3_ERR.M_Ready := FALSE;
   S701_LM_2_CLAMP3_ERR.T_CHK1 := T#0MS;
   S701_LM_2_CLAMP3_ERR.T_CHK2 := T#0MS;
   S701_LM_2_CLAMP3_ERR.PB_Lamp_CHK := FALSE;
   S701_LM_2_CLAMP3_ERR.PB_Error_Rst := FALSE;
   S701_LM_2_CLAMP3_ERR.M_FLICK := FALSE;
   S701_LM_2_CLAMP3_ERR.M_Adv_Err := FALSE;
   S701_LM_2_CLAMP3_ERR.M_Ret_Err := FALSE;
   S701_LM_2_CLAMP3_ERR.LP_Adv := FALSE;
   S701_LM_2_CLAMP3_ERR.LP_Ret := FALSE;
   S701_LM_2_CLAMP3_ERR.Visu_Adv := W#16#0;
   S701_LM_2_CLAMP3_ERR.Visu_Ret := W#16#0;
   S701_LM_2_CLAMP3_ERR.Error_T1.IN := FALSE;
   S701_LM_2_CLAMP3_ERR.Error_T1.PT := T#0MS;
   S701_LM_2_CLAMP3_ERR.Error_T1.Q := FALSE;
   S701_LM_2_CLAMP3_ERR.Error_T1.ET := T#0MS;
   S701_LM_2_CLAMP3_ERR.Error_T1.STATE := B#16#0;
   S701_LM_2_CLAMP3_ERR.Error_T1.STIME := T#0MS;
   S701_LM_2_CLAMP3_ERR.Error_T1.ATIME := T#0MS;
   S701_LM_2_CLAMP3_ERR.Error_T2.IN := FALSE;
   S701_LM_2_CLAMP3_ERR.Error_T2.PT := T#0MS;
   S701_LM_2_CLAMP3_ERR.Error_T2.Q := FALSE;
   S701_LM_2_CLAMP3_ERR.Error_T2.ET := T#0MS;
   S701_LM_2_CLAMP3_ERR.Error_T2.STATE := B#16#0;
   S701_LM_2_CLAMP3_ERR.Error_T2.STIME := T#0MS;
   S701_LM_2_CLAMP3_ERR.Error_T2.ATIME := T#0MS;
   S701_LM_2_CLAMP3_ERR.CHK_Aux1 := FALSE;
   S701_LM_2_CLAMP3_ERR.CHK_Aux2 := FALSE;
   S701_LM_2_CLAMP3_ERR.Error_T1_DN := FALSE;
   S701_LM_2_CLAMP3_ERR.Error_T2_DN := FALSE;
   S701_LM_2_CLAMP3_ERR.Adv_Memo := FALSE;
   S701_LM_2_CLAMP3_ERR.Visu_Adv_Arr[0] := FALSE;
   S701_LM_2_CLAMP3_ERR.Visu_Adv_Arr[1] := FALSE;
   S701_LM_2_CLAMP3_ERR.Visu_Adv_Arr[2] := FALSE;
   S701_LM_2_CLAMP3_ERR.Visu_Adv_Arr[3] := FALSE;
   S701_LM_2_CLAMP3_ERR.Visu_Adv_Arr[4] := FALSE;
   S701_LM_2_CLAMP3_ERR.Visu_Adv_Arr[5] := FALSE;
   S701_LM_2_CLAMP3_ERR.Visu_Adv_Arr[6] := FALSE;
   S701_LM_2_CLAMP3_ERR.Visu_Adv_Arr[7] := FALSE;
   S701_LM_2_CLAMP3_ERR.Visu_Adv_Arr[8] := FALSE;
   S701_LM_2_CLAMP3_ERR.Visu_Adv_Arr[9] := FALSE;
   S701_LM_2_CLAMP3_ERR.Visu_Adv_Arr[10] := FALSE;
   S701_LM_2_CLAMP3_ERR.Visu_Adv_Arr[11] := FALSE;
   S701_LM_2_CLAMP3_ERR.Visu_Adv_Arr[12] := FALSE;
   S701_LM_2_CLAMP3_ERR.Visu_Adv_Arr[13] := FALSE;
   S701_LM_2_CLAMP3_ERR.Visu_Adv_Arr[14] := FALSE;
   S701_LM_2_CLAMP3_ERR.Visu_Adv_Arr[15] := FALSE;
   S701_LM_2_CLAMP3_ERR.Visu_Ret_Arr[0] := FALSE;
   S701_LM_2_CLAMP3_ERR.Visu_Ret_Arr[1] := FALSE;
   S701_LM_2_CLAMP3_ERR.Visu_Ret_Arr[2] := FALSE;
   S701_LM_2_CLAMP3_ERR.Visu_Ret_Arr[3] := FALSE;
   S701_LM_2_CLAMP3_ERR.Visu_Ret_Arr[4] := FALSE;
   S701_LM_2_CLAMP3_ERR.Visu_Ret_Arr[5] := FALSE;
   S701_LM_2_CLAMP3_ERR.Visu_Ret_Arr[6] := FALSE;
   S701_LM_2_CLAMP3_ERR.Visu_Ret_Arr[7] := FALSE;
   S701_LM_2_CLAMP3_ERR.Visu_Ret_Arr[8] := FALSE;
   S701_LM_2_CLAMP3_ERR.Visu_Ret_Arr[9] := FALSE;
   S701_LM_2_CLAMP3_ERR.Visu_Ret_Arr[10] := FALSE;
   S701_LM_2_CLAMP3_ERR.Visu_Ret_Arr[11] := FALSE;
   S701_LM_2_CLAMP3_ERR.Visu_Ret_Arr[12] := FALSE;
   S701_LM_2_CLAMP3_ERR.Visu_Ret_Arr[13] := FALSE;
   S701_LM_2_CLAMP3_ERR.Visu_Ret_Arr[14] := FALSE;
   S701_LM_2_CLAMP3_ERR.Visu_Ret_Arr[15] := FALSE;
   S701_LM_2_CLAMP3_ERR.BLK_Move_Ret := 0;
   S701_LM_2_CLAMP3_ERR.Enable := FALSE;
   S701_LM_2_CLAMP3_ERR.Adv_End := FALSE;
   S701_LM_2_CLAMP3_ERR.Ret_End := FALSE;
   S701_TL_PIN1_ERR.Enable_Aux := FALSE;
   S701_TL_PIN1_ERR.Adv_Amount := 0;
   S701_TL_PIN1_ERR.Ret_Amount := 0;
   S701_TL_PIN1_ERR.LS_Adv1 := FALSE;
   S701_TL_PIN1_ERR.LS_Ret1 := FALSE;
   S701_TL_PIN1_ERR.LS_Adv2 := FALSE;
   S701_TL_PIN1_ERR.LS_Ret2 := FALSE;
   S701_TL_PIN1_ERR.LS_Adv3 := FALSE;
   S701_TL_PIN1_ERR.LS_Ret3 := FALSE;
   S701_TL_PIN1_ERR.LS_Adv4 := FALSE;
   S701_TL_PIN1_ERR.LS_Ret4 := FALSE;
   S701_TL_PIN1_ERR.SOL_Adv := FALSE;
   S701_TL_PIN1_ERR.SOL_Ret := FALSE;
   S701_TL_PIN1_ERR.M_Ready := FALSE;
   S701_TL_PIN1_ERR.T_CHK1 := T#0MS;
   S701_TL_PIN1_ERR.T_CHK2 := T#0MS;
   S701_TL_PIN1_ERR.PB_Lamp_CHK := FALSE;
   S701_TL_PIN1_ERR.PB_Error_Rst := FALSE;
   S701_TL_PIN1_ERR.M_FLICK := FALSE;
   S701_TL_PIN1_ERR.M_Adv_Err := FALSE;
   S701_TL_PIN1_ERR.M_Ret_Err := FALSE;
   S701_TL_PIN1_ERR.LP_Adv := FALSE;
   S701_TL_PIN1_ERR.LP_Ret := FALSE;
   S701_TL_PIN1_ERR.Visu_Adv := W#16#0;
   S701_TL_PIN1_ERR.Visu_Ret := W#16#0;
   S701_TL_PIN1_ERR.Error_T1.IN := FALSE;
   S701_TL_PIN1_ERR.Error_T1.PT := T#0MS;
   S701_TL_PIN1_ERR.Error_T1.Q := FALSE;
   S701_TL_PIN1_ERR.Error_T1.ET := T#0MS;
   S701_TL_PIN1_ERR.Error_T1.STATE := B#16#0;
   S701_TL_PIN1_ERR.Error_T1.STIME := T#0MS;
   S701_TL_PIN1_ERR.Error_T1.ATIME := T#0MS;
   S701_TL_PIN1_ERR.Error_T2.IN := FALSE;
   S701_TL_PIN1_ERR.Error_T2.PT := T#0MS;
   S701_TL_PIN1_ERR.Error_T2.Q := FALSE;
   S701_TL_PIN1_ERR.Error_T2.ET := T#0MS;
   S701_TL_PIN1_ERR.Error_T2.STATE := B#16#0;
   S701_TL_PIN1_ERR.Error_T2.STIME := T#0MS;
   S701_TL_PIN1_ERR.Error_T2.ATIME := T#0MS;
   S701_TL_PIN1_ERR.CHK_Aux1 := FALSE;
   S701_TL_PIN1_ERR.CHK_Aux2 := FALSE;
   S701_TL_PIN1_ERR.Error_T1_DN := FALSE;
   S701_TL_PIN1_ERR.Error_T2_DN := FALSE;
   S701_TL_PIN1_ERR.Adv_Memo := FALSE;
   S701_TL_PIN1_ERR.Visu_Adv_Arr[0] := FALSE;
   S701_TL_PIN1_ERR.Visu_Adv_Arr[1] := FALSE;
   S701_TL_PIN1_ERR.Visu_Adv_Arr[2] := FALSE;
   S701_TL_PIN1_ERR.Visu_Adv_Arr[3] := FALSE;
   S701_TL_PIN1_ERR.Visu_Adv_Arr[4] := FALSE;
   S701_TL_PIN1_ERR.Visu_Adv_Arr[5] := FALSE;
   S701_TL_PIN1_ERR.Visu_Adv_Arr[6] := FALSE;
   S701_TL_PIN1_ERR.Visu_Adv_Arr[7] := FALSE;
   S701_TL_PIN1_ERR.Visu_Adv_Arr[8] := FALSE;
   S701_TL_PIN1_ERR.Visu_Adv_Arr[9] := FALSE;
   S701_TL_PIN1_ERR.Visu_Adv_Arr[10] := FALSE;
   S701_TL_PIN1_ERR.Visu_Adv_Arr[11] := FALSE;
   S701_TL_PIN1_ERR.Visu_Adv_Arr[12] := FALSE;
   S701_TL_PIN1_ERR.Visu_Adv_Arr[13] := FALSE;
   S701_TL_PIN1_ERR.Visu_Adv_Arr[14] := FALSE;
   S701_TL_PIN1_ERR.Visu_Adv_Arr[15] := FALSE;
   S701_TL_PIN1_ERR.Visu_Ret_Arr[0] := FALSE;
   S701_TL_PIN1_ERR.Visu_Ret_Arr[1] := FALSE;
   S701_TL_PIN1_ERR.Visu_Ret_Arr[2] := FALSE;
   S701_TL_PIN1_ERR.Visu_Ret_Arr[3] := FALSE;
   S701_TL_PIN1_ERR.Visu_Ret_Arr[4] := FALSE;
   S701_TL_PIN1_ERR.Visu_Ret_Arr[5] := FALSE;
   S701_TL_PIN1_ERR.Visu_Ret_Arr[6] := FALSE;
   S701_TL_PIN1_ERR.Visu_Ret_Arr[7] := FALSE;
   S701_TL_PIN1_ERR.Visu_Ret_Arr[8] := FALSE;
   S701_TL_PIN1_ERR.Visu_Ret_Arr[9] := FALSE;
   S701_TL_PIN1_ERR.Visu_Ret_Arr[10] := FALSE;
   S701_TL_PIN1_ERR.Visu_Ret_Arr[11] := FALSE;
   S701_TL_PIN1_ERR.Visu_Ret_Arr[12] := FALSE;
   S701_TL_PIN1_ERR.Visu_Ret_Arr[13] := FALSE;
   S701_TL_PIN1_ERR.Visu_Ret_Arr[14] := FALSE;
   S701_TL_PIN1_ERR.Visu_Ret_Arr[15] := FALSE;
   S701_TL_PIN1_ERR.BLK_Move_Ret := 0;
   S701_TL_PIN1_ERR.Enable := FALSE;
   S701_TL_PIN1_ERR.Adv_End := FALSE;
   S701_TL_PIN1_ERR.Ret_End := FALSE;
   S701_LM_2_CLAMP4_ERR.Enable_Aux := FALSE;
   S701_LM_2_CLAMP4_ERR.Adv_Amount := 0;
   S701_LM_2_CLAMP4_ERR.Ret_Amount := 0;
   S701_LM_2_CLAMP4_ERR.LS_Adv1 := FALSE;
   S701_LM_2_CLAMP4_ERR.LS_Ret1 := FALSE;
   S701_LM_2_CLAMP4_ERR.LS_Adv2 := FALSE;
   S701_LM_2_CLAMP4_ERR.LS_Ret2 := FALSE;
   S701_LM_2_CLAMP4_ERR.LS_Adv3 := FALSE;
   S701_LM_2_CLAMP4_ERR.LS_Ret3 := FALSE;
   S701_LM_2_CLAMP4_ERR.LS_Adv4 := FALSE;
   S701_LM_2_CLAMP4_ERR.LS_Ret4 := FALSE;
   S701_LM_2_CLAMP4_ERR.SOL_Adv := FALSE;
   S701_LM_2_CLAMP4_ERR.SOL_Ret := FALSE;
   S701_LM_2_CLAMP4_ERR.M_Ready := FALSE;
   S701_LM_2_CLAMP4_ERR.T_CHK1 := T#0MS;
   S701_LM_2_CLAMP4_ERR.T_CHK2 := T#0MS;
   S701_LM_2_CLAMP4_ERR.PB_Lamp_CHK := FALSE;
   S701_LM_2_CLAMP4_ERR.PB_Error_Rst := FALSE;
   S701_LM_2_CLAMP4_ERR.M_FLICK := FALSE;
   S701_LM_2_CLAMP4_ERR.M_Adv_Err := FALSE;
   S701_LM_2_CLAMP4_ERR.M_Ret_Err := FALSE;
   S701_LM_2_CLAMP4_ERR.LP_Adv := FALSE;
   S701_LM_2_CLAMP4_ERR.LP_Ret := FALSE;
   S701_LM_2_CLAMP4_ERR.Visu_Adv := W#16#0;
   S701_LM_2_CLAMP4_ERR.Visu_Ret := W#16#0;
   S701_LM_2_CLAMP4_ERR.Error_T1.IN := FALSE;
   S701_LM_2_CLAMP4_ERR.Error_T1.PT := T#0MS;
   S701_LM_2_CLAMP4_ERR.Error_T1.Q := FALSE;
   S701_LM_2_CLAMP4_ERR.Error_T1.ET := T#0MS;
   S701_LM_2_CLAMP4_ERR.Error_T1.STATE := B#16#0;
   S701_LM_2_CLAMP4_ERR.Error_T1.STIME := T#0MS;
   S701_LM_2_CLAMP4_ERR.Error_T1.ATIME := T#0MS;
   S701_LM_2_CLAMP4_ERR.Error_T2.IN := FALSE;
   S701_LM_2_CLAMP4_ERR.Error_T2.PT := T#0MS;
   S701_LM_2_CLAMP4_ERR.Error_T2.Q := FALSE;
   S701_LM_2_CLAMP4_ERR.Error_T2.ET := T#0MS;
   S701_LM_2_CLAMP4_ERR.Error_T2.STATE := B#16#0;
   S701_LM_2_CLAMP4_ERR.Error_T2.STIME := T#0MS;
   S701_LM_2_CLAMP4_ERR.Error_T2.ATIME := T#0MS;
   S701_LM_2_CLAMP4_ERR.CHK_Aux1 := FALSE;
   S701_LM_2_CLAMP4_ERR.CHK_Aux2 := FALSE;
   S701_LM_2_CLAMP4_ERR.Error_T1_DN := FALSE;
   S701_LM_2_CLAMP4_ERR.Error_T2_DN := FALSE;
   S701_LM_2_CLAMP4_ERR.Adv_Memo := FALSE;
   S701_LM_2_CLAMP4_ERR.Visu_Adv_Arr[0] := FALSE;
   S701_LM_2_CLAMP4_ERR.Visu_Adv_Arr[1] := FALSE;
   S701_LM_2_CLAMP4_ERR.Visu_Adv_Arr[2] := FALSE;
   S701_LM_2_CLAMP4_ERR.Visu_Adv_Arr[3] := FALSE;
   S701_LM_2_CLAMP4_ERR.Visu_Adv_Arr[4] := FALSE;
   S701_LM_2_CLAMP4_ERR.Visu_Adv_Arr[5] := FALSE;
   S701_LM_2_CLAMP4_ERR.Visu_Adv_Arr[6] := FALSE;
   S701_LM_2_CLAMP4_ERR.Visu_Adv_Arr[7] := FALSE;
   S701_LM_2_CLAMP4_ERR.Visu_Adv_Arr[8] := FALSE;
   S701_LM_2_CLAMP4_ERR.Visu_Adv_Arr[9] := FALSE;
   S701_LM_2_CLAMP4_ERR.Visu_Adv_Arr[10] := FALSE;
   S701_LM_2_CLAMP4_ERR.Visu_Adv_Arr[11] := FALSE;
   S701_LM_2_CLAMP4_ERR.Visu_Adv_Arr[12] := FALSE;
   S701_LM_2_CLAMP4_ERR.Visu_Adv_Arr[13] := FALSE;
   S701_LM_2_CLAMP4_ERR.Visu_Adv_Arr[14] := FALSE;
   S701_LM_2_CLAMP4_ERR.Visu_Adv_Arr[15] := FALSE;
   S701_LM_2_CLAMP4_ERR.Visu_Ret_Arr[0] := FALSE;
   S701_LM_2_CLAMP4_ERR.Visu_Ret_Arr[1] := FALSE;
   S701_LM_2_CLAMP4_ERR.Visu_Ret_Arr[2] := FALSE;
   S701_LM_2_CLAMP4_ERR.Visu_Ret_Arr[3] := FALSE;
   S701_LM_2_CLAMP4_ERR.Visu_Ret_Arr[4] := FALSE;
   S701_LM_2_CLAMP4_ERR.Visu_Ret_Arr[5] := FALSE;
   S701_LM_2_CLAMP4_ERR.Visu_Ret_Arr[6] := FALSE;
   S701_LM_2_CLAMP4_ERR.Visu_Ret_Arr[7] := FALSE;
   S701_LM_2_CLAMP4_ERR.Visu_Ret_Arr[8] := FALSE;
   S701_LM_2_CLAMP4_ERR.Visu_Ret_Arr[9] := FALSE;
   S701_LM_2_CLAMP4_ERR.Visu_Ret_Arr[10] := FALSE;
   S701_LM_2_CLAMP4_ERR.Visu_Ret_Arr[11] := FALSE;
   S701_LM_2_CLAMP4_ERR.Visu_Ret_Arr[12] := FALSE;
   S701_LM_2_CLAMP4_ERR.Visu_Ret_Arr[13] := FALSE;
   S701_LM_2_CLAMP4_ERR.Visu_Ret_Arr[14] := FALSE;
   S701_LM_2_CLAMP4_ERR.Visu_Ret_Arr[15] := FALSE;
   S701_LM_2_CLAMP4_ERR.BLK_Move_Ret := 0;
   S701_LM_2_CLAMP4_ERR.Enable := FALSE;
   S701_LM_2_CLAMP4_ERR.Adv_End := FALSE;
   S701_LM_2_CLAMP4_ERR.Ret_End := FALSE;
   S701_LM_2_CLAMP5_ERR.Enable_Aux := FALSE;
   S701_LM_2_CLAMP5_ERR.Adv_Amount := 0;
   S701_LM_2_CLAMP5_ERR.Ret_Amount := 0;
   S701_LM_2_CLAMP5_ERR.LS_Adv1 := FALSE;
   S701_LM_2_CLAMP5_ERR.LS_Ret1 := FALSE;
   S701_LM_2_CLAMP5_ERR.LS_Adv2 := FALSE;
   S701_LM_2_CLAMP5_ERR.LS_Ret2 := FALSE;
   S701_LM_2_CLAMP5_ERR.LS_Adv3 := FALSE;
   S701_LM_2_CLAMP5_ERR.LS_Ret3 := FALSE;
   S701_LM_2_CLAMP5_ERR.LS_Adv4 := FALSE;
   S701_LM_2_CLAMP5_ERR.LS_Ret4 := FALSE;
   S701_LM_2_CLAMP5_ERR.SOL_Adv := FALSE;
   S701_LM_2_CLAMP5_ERR.SOL_Ret := FALSE;
   S701_LM_2_CLAMP5_ERR.M_Ready := FALSE;
   S701_LM_2_CLAMP5_ERR.T_CHK1 := T#0MS;
   S701_LM_2_CLAMP5_ERR.T_CHK2 := T#0MS;
   S701_LM_2_CLAMP5_ERR.PB_Lamp_CHK := FALSE;
   S701_LM_2_CLAMP5_ERR.PB_Error_Rst := FALSE;
   S701_LM_2_CLAMP5_ERR.M_FLICK := FALSE;
   S701_LM_2_CLAMP5_ERR.M_Adv_Err := FALSE;
   S701_LM_2_CLAMP5_ERR.M_Ret_Err := FALSE;
   S701_LM_2_CLAMP5_ERR.LP_Adv := FALSE;
   S701_LM_2_CLAMP5_ERR.LP_Ret := FALSE;
   S701_LM_2_CLAMP5_ERR.Visu_Adv := W#16#0;
   S701_LM_2_CLAMP5_ERR.Visu_Ret := W#16#0;
   S701_LM_2_CLAMP5_ERR.Error_T1.IN := FALSE;
   S701_LM_2_CLAMP5_ERR.Error_T1.PT := T#0MS;
   S701_LM_2_CLAMP5_ERR.Error_T1.Q := FALSE;
   S701_LM_2_CLAMP5_ERR.Error_T1.ET := T#0MS;
   S701_LM_2_CLAMP5_ERR.Error_T1.STATE := B#16#0;
   S701_LM_2_CLAMP5_ERR.Error_T1.STIME := T#0MS;
   S701_LM_2_CLAMP5_ERR.Error_T1.ATIME := T#0MS;
   S701_LM_2_CLAMP5_ERR.Error_T2.IN := FALSE;
   S701_LM_2_CLAMP5_ERR.Error_T2.PT := T#0MS;
   S701_LM_2_CLAMP5_ERR.Error_T2.Q := FALSE;
   S701_LM_2_CLAMP5_ERR.Error_T2.ET := T#0MS;
   S701_LM_2_CLAMP5_ERR.Error_T2.STATE := B#16#0;
   S701_LM_2_CLAMP5_ERR.Error_T2.STIME := T#0MS;
   S701_LM_2_CLAMP5_ERR.Error_T2.ATIME := T#0MS;
   S701_LM_2_CLAMP5_ERR.CHK_Aux1 := FALSE;
   S701_LM_2_CLAMP5_ERR.CHK_Aux2 := FALSE;
   S701_LM_2_CLAMP5_ERR.Error_T1_DN := FALSE;
   S701_LM_2_CLAMP5_ERR.Error_T2_DN := FALSE;
   S701_LM_2_CLAMP5_ERR.Adv_Memo := FALSE;
   S701_LM_2_CLAMP5_ERR.Visu_Adv_Arr[0] := FALSE;
   S701_LM_2_CLAMP5_ERR.Visu_Adv_Arr[1] := FALSE;
   S701_LM_2_CLAMP5_ERR.Visu_Adv_Arr[2] := FALSE;
   S701_LM_2_CLAMP5_ERR.Visu_Adv_Arr[3] := FALSE;
   S701_LM_2_CLAMP5_ERR.Visu_Adv_Arr[4] := FALSE;
   S701_LM_2_CLAMP5_ERR.Visu_Adv_Arr[5] := FALSE;
   S701_LM_2_CLAMP5_ERR.Visu_Adv_Arr[6] := FALSE;
   S701_LM_2_CLAMP5_ERR.Visu_Adv_Arr[7] := FALSE;
   S701_LM_2_CLAMP5_ERR.Visu_Adv_Arr[8] := FALSE;
   S701_LM_2_CLAMP5_ERR.Visu_Adv_Arr[9] := FALSE;
   S701_LM_2_CLAMP5_ERR.Visu_Adv_Arr[10] := FALSE;
   S701_LM_2_CLAMP5_ERR.Visu_Adv_Arr[11] := FALSE;
   S701_LM_2_CLAMP5_ERR.Visu_Adv_Arr[12] := FALSE;
   S701_LM_2_CLAMP5_ERR.Visu_Adv_Arr[13] := FALSE;
   S701_LM_2_CLAMP5_ERR.Visu_Adv_Arr[14] := FALSE;
   S701_LM_2_CLAMP5_ERR.Visu_Adv_Arr[15] := FALSE;
   S701_LM_2_CLAMP5_ERR.Visu_Ret_Arr[0] := FALSE;
   S701_LM_2_CLAMP5_ERR.Visu_Ret_Arr[1] := FALSE;
   S701_LM_2_CLAMP5_ERR.Visu_Ret_Arr[2] := FALSE;
   S701_LM_2_CLAMP5_ERR.Visu_Ret_Arr[3] := FALSE;
   S701_LM_2_CLAMP5_ERR.Visu_Ret_Arr[4] := FALSE;
   S701_LM_2_CLAMP5_ERR.Visu_Ret_Arr[5] := FALSE;
   S701_LM_2_CLAMP5_ERR.Visu_Ret_Arr[6] := FALSE;
   S701_LM_2_CLAMP5_ERR.Visu_Ret_Arr[7] := FALSE;
   S701_LM_2_CLAMP5_ERR.Visu_Ret_Arr[8] := FALSE;
   S701_LM_2_CLAMP5_ERR.Visu_Ret_Arr[9] := FALSE;
   S701_LM_2_CLAMP5_ERR.Visu_Ret_Arr[10] := FALSE;
   S701_LM_2_CLAMP5_ERR.Visu_Ret_Arr[11] := FALSE;
   S701_LM_2_CLAMP5_ERR.Visu_Ret_Arr[12] := FALSE;
   S701_LM_2_CLAMP5_ERR.Visu_Ret_Arr[13] := FALSE;
   S701_LM_2_CLAMP5_ERR.Visu_Ret_Arr[14] := FALSE;
   S701_LM_2_CLAMP5_ERR.Visu_Ret_Arr[15] := FALSE;
   S701_LM_2_CLAMP5_ERR.BLK_Move_Ret := 0;
   S701_LM_2_CLAMP5_ERR.Enable := FALSE;
   S701_LM_2_CLAMP5_ERR.Adv_End := FALSE;
   S701_LM_2_CLAMP5_ERR.Ret_End := FALSE;
   S701_LM_FDR_SFT_ERR.Enable_Aux := FALSE;
   S701_LM_FDR_SFT_ERR.Adv_Amount := 0;
   S701_LM_FDR_SFT_ERR.Ret_Amount := 0;
   S701_LM_FDR_SFT_ERR.LS_Adv1 := FALSE;
   S701_LM_FDR_SFT_ERR.LS_Ret1 := FALSE;
   S701_LM_FDR_SFT_ERR.LS_Adv2 := FALSE;
   S701_LM_FDR_SFT_ERR.LS_Ret2 := FALSE;
   S701_LM_FDR_SFT_ERR.LS_Adv3 := FALSE;
   S701_LM_FDR_SFT_ERR.LS_Ret3 := FALSE;
   S701_LM_FDR_SFT_ERR.LS_Adv4 := FALSE;
   S701_LM_FDR_SFT_ERR.LS_Ret4 := FALSE;
   S701_LM_FDR_SFT_ERR.SOL_Adv := FALSE;
   S701_LM_FDR_SFT_ERR.SOL_Ret := FALSE;
   S701_LM_FDR_SFT_ERR.M_Ready := FALSE;
   S701_LM_FDR_SFT_ERR.T_CHK1 := T#0MS;
   S701_LM_FDR_SFT_ERR.T_CHK2 := T#0MS;
   S701_LM_FDR_SFT_ERR.PB_Lamp_CHK := FALSE;
   S701_LM_FDR_SFT_ERR.PB_Error_Rst := FALSE;
   S701_LM_FDR_SFT_ERR.M_FLICK := FALSE;
   S701_LM_FDR_SFT_ERR.M_Adv_Err := FALSE;
   S701_LM_FDR_SFT_ERR.M_Ret_Err := FALSE;
   S701_LM_FDR_SFT_ERR.LP_Adv := FALSE;
   S701_LM_FDR_SFT_ERR.LP_Ret := FALSE;
   S701_LM_FDR_SFT_ERR.Visu_Adv := W#16#0;
   S701_LM_FDR_SFT_ERR.Visu_Ret := W#16#0;
   S701_LM_FDR_SFT_ERR.Error_T1.IN := FALSE;
   S701_LM_FDR_SFT_ERR.Error_T1.PT := T#0MS;
   S701_LM_FDR_SFT_ERR.Error_T1.Q := FALSE;
   S701_LM_FDR_SFT_ERR.Error_T1.ET := T#0MS;
   S701_LM_FDR_SFT_ERR.Error_T1.STATE := B#16#0;
   S701_LM_FDR_SFT_ERR.Error_T1.STIME := T#0MS;
   S701_LM_FDR_SFT_ERR.Error_T1.ATIME := T#0MS;
   S701_LM_FDR_SFT_ERR.Error_T2.IN := FALSE;
   S701_LM_FDR_SFT_ERR.Error_T2.PT := T#0MS;
   S701_LM_FDR_SFT_ERR.Error_T2.Q := FALSE;
   S701_LM_FDR_SFT_ERR.Error_T2.ET := T#0MS;
   S701_LM_FDR_SFT_ERR.Error_T2.STATE := B#16#0;
   S701_LM_FDR_SFT_ERR.Error_T2.STIME := T#0MS;
   S701_LM_FDR_SFT_ERR.Error_T2.ATIME := T#0MS;
   S701_LM_FDR_SFT_ERR.CHK_Aux1 := FALSE;
   S701_LM_FDR_SFT_ERR.CHK_Aux2 := FALSE;
   S701_LM_FDR_SFT_ERR.Error_T1_DN := FALSE;
   S701_LM_FDR_SFT_ERR.Error_T2_DN := FALSE;
   S701_LM_FDR_SFT_ERR.Adv_Memo := FALSE;
   S701_LM_FDR_SFT_ERR.Visu_Adv_Arr[0] := FALSE;
   S701_LM_FDR_SFT_ERR.Visu_Adv_Arr[1] := FALSE;
   S701_LM_FDR_SFT_ERR.Visu_Adv_Arr[2] := FALSE;
   S701_LM_FDR_SFT_ERR.Visu_Adv_Arr[3] := FALSE;
   S701_LM_FDR_SFT_ERR.Visu_Adv_Arr[4] := FALSE;
   S701_LM_FDR_SFT_ERR.Visu_Adv_Arr[5] := FALSE;
   S701_LM_FDR_SFT_ERR.Visu_Adv_Arr[6] := FALSE;
   S701_LM_FDR_SFT_ERR.Visu_Adv_Arr[7] := FALSE;
   S701_LM_FDR_SFT_ERR.Visu_Adv_Arr[8] := FALSE;
   S701_LM_FDR_SFT_ERR.Visu_Adv_Arr[9] := FALSE;
   S701_LM_FDR_SFT_ERR.Visu_Adv_Arr[10] := FALSE;
   S701_LM_FDR_SFT_ERR.Visu_Adv_Arr[11] := FALSE;
   S701_LM_FDR_SFT_ERR.Visu_Adv_Arr[12] := FALSE;
   S701_LM_FDR_SFT_ERR.Visu_Adv_Arr[13] := FALSE;
   S701_LM_FDR_SFT_ERR.Visu_Adv_Arr[14] := FALSE;
   S701_LM_FDR_SFT_ERR.Visu_Adv_Arr[15] := FALSE;
   S701_LM_FDR_SFT_ERR.Visu_Ret_Arr[0] := FALSE;
   S701_LM_FDR_SFT_ERR.Visu_Ret_Arr[1] := FALSE;
   S701_LM_FDR_SFT_ERR.Visu_Ret_Arr[2] := FALSE;
   S701_LM_FDR_SFT_ERR.Visu_Ret_Arr[3] := FALSE;
   S701_LM_FDR_SFT_ERR.Visu_Ret_Arr[4] := FALSE;
   S701_LM_FDR_SFT_ERR.Visu_Ret_Arr[5] := FALSE;
   S701_LM_FDR_SFT_ERR.Visu_Ret_Arr[6] := FALSE;
   S701_LM_FDR_SFT_ERR.Visu_Ret_Arr[7] := FALSE;
   S701_LM_FDR_SFT_ERR.Visu_Ret_Arr[8] := FALSE;
   S701_LM_FDR_SFT_ERR.Visu_Ret_Arr[9] := FALSE;
   S701_LM_FDR_SFT_ERR.Visu_Ret_Arr[10] := FALSE;
   S701_LM_FDR_SFT_ERR.Visu_Ret_Arr[11] := FALSE;
   S701_LM_FDR_SFT_ERR.Visu_Ret_Arr[12] := FALSE;
   S701_LM_FDR_SFT_ERR.Visu_Ret_Arr[13] := FALSE;
   S701_LM_FDR_SFT_ERR.Visu_Ret_Arr[14] := FALSE;
   S701_LM_FDR_SFT_ERR.Visu_Ret_Arr[15] := FALSE;
   S701_LM_FDR_SFT_ERR.BLK_Move_Ret := 0;
   S701_LM_FDR_SFT_ERR.Enable := FALSE;
   S701_LM_FDR_SFT_ERR.Adv_End := FALSE;
   S701_LM_FDR_SFT_ERR.Ret_End := FALSE;
   S701_LM_FDR_PIN_ERR.Enable_Aux := FALSE;
   S701_LM_FDR_PIN_ERR.Adv_Amount := 0;
   S701_LM_FDR_PIN_ERR.Ret_Amount := 0;
   S701_LM_FDR_PIN_ERR.LS_Adv1 := FALSE;
   S701_LM_FDR_PIN_ERR.LS_Ret1 := FALSE;
   S701_LM_FDR_PIN_ERR.LS_Adv2 := FALSE;
   S701_LM_FDR_PIN_ERR.LS_Ret2 := FALSE;
   S701_LM_FDR_PIN_ERR.LS_Adv3 := FALSE;
   S701_LM_FDR_PIN_ERR.LS_Ret3 := FALSE;
   S701_LM_FDR_PIN_ERR.LS_Adv4 := FALSE;
   S701_LM_FDR_PIN_ERR.LS_Ret4 := FALSE;
   S701_LM_FDR_PIN_ERR.SOL_Adv := FALSE;
   S701_LM_FDR_PIN_ERR.SOL_Ret := FALSE;
   S701_LM_FDR_PIN_ERR.M_Ready := FALSE;
   S701_LM_FDR_PIN_ERR.T_CHK1 := T#0MS;
   S701_LM_FDR_PIN_ERR.T_CHK2 := T#0MS;
   S701_LM_FDR_PIN_ERR.PB_Lamp_CHK := FALSE;
   S701_LM_FDR_PIN_ERR.PB_Error_Rst := FALSE;
   S701_LM_FDR_PIN_ERR.M_FLICK := FALSE;
   S701_LM_FDR_PIN_ERR.M_Adv_Err := FALSE;
   S701_LM_FDR_PIN_ERR.M_Ret_Err := FALSE;
   S701_LM_FDR_PIN_ERR.LP_Adv := FALSE;
   S701_LM_FDR_PIN_ERR.LP_Ret := FALSE;
   S701_LM_FDR_PIN_ERR.Visu_Adv := W#16#0;
   S701_LM_FDR_PIN_ERR.Visu_Ret := W#16#0;
   S701_LM_FDR_PIN_ERR.Error_T1.IN := FALSE;
   S701_LM_FDR_PIN_ERR.Error_T1.PT := T#0MS;
   S701_LM_FDR_PIN_ERR.Error_T1.Q := FALSE;
   S701_LM_FDR_PIN_ERR.Error_T1.ET := T#0MS;
   S701_LM_FDR_PIN_ERR.Error_T1.STATE := B#16#0;
   S701_LM_FDR_PIN_ERR.Error_T1.STIME := T#0MS;
   S701_LM_FDR_PIN_ERR.Error_T1.ATIME := T#0MS;
   S701_LM_FDR_PIN_ERR.Error_T2.IN := FALSE;
   S701_LM_FDR_PIN_ERR.Error_T2.PT := T#0MS;
   S701_LM_FDR_PIN_ERR.Error_T2.Q := FALSE;
   S701_LM_FDR_PIN_ERR.Error_T2.ET := T#0MS;
   S701_LM_FDR_PIN_ERR.Error_T2.STATE := B#16#0;
   S701_LM_FDR_PIN_ERR.Error_T2.STIME := T#0MS;
   S701_LM_FDR_PIN_ERR.Error_T2.ATIME := T#0MS;
   S701_LM_FDR_PIN_ERR.CHK_Aux1 := FALSE;
   S701_LM_FDR_PIN_ERR.CHK_Aux2 := FALSE;
   S701_LM_FDR_PIN_ERR.Error_T1_DN := FALSE;
   S701_LM_FDR_PIN_ERR.Error_T2_DN := FALSE;
   S701_LM_FDR_PIN_ERR.Adv_Memo := FALSE;
   S701_LM_FDR_PIN_ERR.Visu_Adv_Arr[0] := FALSE;
   S701_LM_FDR_PIN_ERR.Visu_Adv_Arr[1] := FALSE;
   S701_LM_FDR_PIN_ERR.Visu_Adv_Arr[2] := FALSE;
   S701_LM_FDR_PIN_ERR.Visu_Adv_Arr[3] := FALSE;
   S701_LM_FDR_PIN_ERR.Visu_Adv_Arr[4] := FALSE;
   S701_LM_FDR_PIN_ERR.Visu_Adv_Arr[5] := FALSE;
   S701_LM_FDR_PIN_ERR.Visu_Adv_Arr[6] := FALSE;
   S701_LM_FDR_PIN_ERR.Visu_Adv_Arr[7] := FALSE;
   S701_LM_FDR_PIN_ERR.Visu_Adv_Arr[8] := FALSE;
   S701_LM_FDR_PIN_ERR.Visu_Adv_Arr[9] := FALSE;
   S701_LM_FDR_PIN_ERR.Visu_Adv_Arr[10] := FALSE;
   S701_LM_FDR_PIN_ERR.Visu_Adv_Arr[11] := FALSE;
   S701_LM_FDR_PIN_ERR.Visu_Adv_Arr[12] := FALSE;
   S701_LM_FDR_PIN_ERR.Visu_Adv_Arr[13] := FALSE;
   S701_LM_FDR_PIN_ERR.Visu_Adv_Arr[14] := FALSE;
   S701_LM_FDR_PIN_ERR.Visu_Adv_Arr[15] := FALSE;
   S701_LM_FDR_PIN_ERR.Visu_Ret_Arr[0] := FALSE;
   S701_LM_FDR_PIN_ERR.Visu_Ret_Arr[1] := FALSE;
   S701_LM_FDR_PIN_ERR.Visu_Ret_Arr[2] := FALSE;
   S701_LM_FDR_PIN_ERR.Visu_Ret_Arr[3] := FALSE;
   S701_LM_FDR_PIN_ERR.Visu_Ret_Arr[4] := FALSE;
   S701_LM_FDR_PIN_ERR.Visu_Ret_Arr[5] := FALSE;
   S701_LM_FDR_PIN_ERR.Visu_Ret_Arr[6] := FALSE;
   S701_LM_FDR_PIN_ERR.Visu_Ret_Arr[7] := FALSE;
   S701_LM_FDR_PIN_ERR.Visu_Ret_Arr[8] := FALSE;
   S701_LM_FDR_PIN_ERR.Visu_Ret_Arr[9] := FALSE;
   S701_LM_FDR_PIN_ERR.Visu_Ret_Arr[10] := FALSE;
   S701_LM_FDR_PIN_ERR.Visu_Ret_Arr[11] := FALSE;
   S701_LM_FDR_PIN_ERR.Visu_Ret_Arr[12] := FALSE;
   S701_LM_FDR_PIN_ERR.Visu_Ret_Arr[13] := FALSE;
   S701_LM_FDR_PIN_ERR.Visu_Ret_Arr[14] := FALSE;
   S701_LM_FDR_PIN_ERR.Visu_Ret_Arr[15] := FALSE;
   S701_LM_FDR_PIN_ERR.BLK_Move_Ret := 0;
   S701_LM_FDR_PIN_ERR.Enable := FALSE;
   S701_LM_FDR_PIN_ERR.Adv_End := FALSE;
   S701_LM_FDR_PIN_ERR.Ret_End := FALSE;
   S701_TL_PIN2_ERR.Enable_Aux := FALSE;
   S701_TL_PIN2_ERR.Adv_Amount := 0;
   S701_TL_PIN2_ERR.Ret_Amount := 0;
   S701_TL_PIN2_ERR.LS_Adv1 := FALSE;
   S701_TL_PIN2_ERR.LS_Ret1 := FALSE;
   S701_TL_PIN2_ERR.LS_Adv2 := FALSE;
   S701_TL_PIN2_ERR.LS_Ret2 := FALSE;
   S701_TL_PIN2_ERR.LS_Adv3 := FALSE;
   S701_TL_PIN2_ERR.LS_Ret3 := FALSE;
   S701_TL_PIN2_ERR.LS_Adv4 := FALSE;
   S701_TL_PIN2_ERR.LS_Ret4 := FALSE;
   S701_TL_PIN2_ERR.SOL_Adv := FALSE;
   S701_TL_PIN2_ERR.SOL_Ret := FALSE;
   S701_TL_PIN2_ERR.M_Ready := FALSE;
   S701_TL_PIN2_ERR.T_CHK1 := T#0MS;
   S701_TL_PIN2_ERR.T_CHK2 := T#0MS;
   S701_TL_PIN2_ERR.PB_Lamp_CHK := FALSE;
   S701_TL_PIN2_ERR.PB_Error_Rst := FALSE;
   S701_TL_PIN2_ERR.M_FLICK := FALSE;
   S701_TL_PIN2_ERR.M_Adv_Err := FALSE;
   S701_TL_PIN2_ERR.M_Ret_Err := FALSE;
   S701_TL_PIN2_ERR.LP_Adv := FALSE;
   S701_TL_PIN2_ERR.LP_Ret := FALSE;
   S701_TL_PIN2_ERR.Visu_Adv := W#16#0;
   S701_TL_PIN2_ERR.Visu_Ret := W#16#0;
   S701_TL_PIN2_ERR.Error_T1.IN := FALSE;
   S701_TL_PIN2_ERR.Error_T1.PT := T#0MS;
   S701_TL_PIN2_ERR.Error_T1.Q := FALSE;
   S701_TL_PIN2_ERR.Error_T1.ET := T#0MS;
   S701_TL_PIN2_ERR.Error_T1.STATE := B#16#0;
   S701_TL_PIN2_ERR.Error_T1.STIME := T#0MS;
   S701_TL_PIN2_ERR.Error_T1.ATIME := T#0MS;
   S701_TL_PIN2_ERR.Error_T2.IN := FALSE;
   S701_TL_PIN2_ERR.Error_T2.PT := T#0MS;
   S701_TL_PIN2_ERR.Error_T2.Q := FALSE;
   S701_TL_PIN2_ERR.Error_T2.ET := T#0MS;
   S701_TL_PIN2_ERR.Error_T2.STATE := B#16#0;
   S701_TL_PIN2_ERR.Error_T2.STIME := T#0MS;
   S701_TL_PIN2_ERR.Error_T2.ATIME := T#0MS;
   S701_TL_PIN2_ERR.CHK_Aux1 := FALSE;
   S701_TL_PIN2_ERR.CHK_Aux2 := FALSE;
   S701_TL_PIN2_ERR.Error_T1_DN := FALSE;
   S701_TL_PIN2_ERR.Error_T2_DN := FALSE;
   S701_TL_PIN2_ERR.Adv_Memo := FALSE;
   S701_TL_PIN2_ERR.Visu_Adv_Arr[0] := FALSE;
   S701_TL_PIN2_ERR.Visu_Adv_Arr[1] := FALSE;
   S701_TL_PIN2_ERR.Visu_Adv_Arr[2] := FALSE;
   S701_TL_PIN2_ERR.Visu_Adv_Arr[3] := FALSE;
   S701_TL_PIN2_ERR.Visu_Adv_Arr[4] := FALSE;
   S701_TL_PIN2_ERR.Visu_Adv_Arr[5] := FALSE;
   S701_TL_PIN2_ERR.Visu_Adv_Arr[6] := FALSE;
   S701_TL_PIN2_ERR.Visu_Adv_Arr[7] := FALSE;
   S701_TL_PIN2_ERR.Visu_Adv_Arr[8] := FALSE;
   S701_TL_PIN2_ERR.Visu_Adv_Arr[9] := FALSE;
   S701_TL_PIN2_ERR.Visu_Adv_Arr[10] := FALSE;
   S701_TL_PIN2_ERR.Visu_Adv_Arr[11] := FALSE;
   S701_TL_PIN2_ERR.Visu_Adv_Arr[12] := FALSE;
   S701_TL_PIN2_ERR.Visu_Adv_Arr[13] := FALSE;
   S701_TL_PIN2_ERR.Visu_Adv_Arr[14] := FALSE;
   S701_TL_PIN2_ERR.Visu_Adv_Arr[15] := FALSE;
   S701_TL_PIN2_ERR.Visu_Ret_Arr[0] := FALSE;
   S701_TL_PIN2_ERR.Visu_Ret_Arr[1] := FALSE;
   S701_TL_PIN2_ERR.Visu_Ret_Arr[2] := FALSE;
   S701_TL_PIN2_ERR.Visu_Ret_Arr[3] := FALSE;
   S701_TL_PIN2_ERR.Visu_Ret_Arr[4] := FALSE;
   S701_TL_PIN2_ERR.Visu_Ret_Arr[5] := FALSE;
   S701_TL_PIN2_ERR.Visu_Ret_Arr[6] := FALSE;
   S701_TL_PIN2_ERR.Visu_Ret_Arr[7] := FALSE;
   S701_TL_PIN2_ERR.Visu_Ret_Arr[8] := FALSE;
   S701_TL_PIN2_ERR.Visu_Ret_Arr[9] := FALSE;
   S701_TL_PIN2_ERR.Visu_Ret_Arr[10] := FALSE;
   S701_TL_PIN2_ERR.Visu_Ret_Arr[11] := FALSE;
   S701_TL_PIN2_ERR.Visu_Ret_Arr[12] := FALSE;
   S701_TL_PIN2_ERR.Visu_Ret_Arr[13] := FALSE;
   S701_TL_PIN2_ERR.Visu_Ret_Arr[14] := FALSE;
   S701_TL_PIN2_ERR.Visu_Ret_Arr[15] := FALSE;
   S701_TL_PIN2_ERR.BLK_Move_Ret := 0;
   S701_TL_PIN2_ERR.Enable := FALSE;
   S701_TL_PIN2_ERR.Adv_End := FALSE;
   S701_TL_PIN2_ERR.Ret_End := FALSE;
   S701_TL_LOCATE1_ERR.Enable_Aux := FALSE;
   S701_TL_LOCATE1_ERR.Adv_Amount := 0;
   S701_TL_LOCATE1_ERR.Ret_Amount := 0;
   S701_TL_LOCATE1_ERR.LS_Adv1 := FALSE;
   S701_TL_LOCATE1_ERR.LS_Ret1 := FALSE;
   S701_TL_LOCATE1_ERR.LS_Adv2 := FALSE;
   S701_TL_LOCATE1_ERR.LS_Ret2 := FALSE;
   S701_TL_LOCATE1_ERR.LS_Adv3 := FALSE;
   S701_TL_LOCATE1_ERR.LS_Ret3 := FALSE;
   S701_TL_LOCATE1_ERR.LS_Adv4 := FALSE;
   S701_TL_LOCATE1_ERR.LS_Ret4 := FALSE;
   S701_TL_LOCATE1_ERR.SOL_Adv := FALSE;
   S701_TL_LOCATE1_ERR.SOL_Ret := FALSE;
   S701_TL_LOCATE1_ERR.M_Ready := FALSE;
   S701_TL_LOCATE1_ERR.T_CHK1 := T#0MS;
   S701_TL_LOCATE1_ERR.T_CHK2 := T#0MS;
   S701_TL_LOCATE1_ERR.PB_Lamp_CHK := FALSE;
   S701_TL_LOCATE1_ERR.PB_Error_Rst := FALSE;
   S701_TL_LOCATE1_ERR.M_FLICK := FALSE;
   S701_TL_LOCATE1_ERR.M_Adv_Err := FALSE;
   S701_TL_LOCATE1_ERR.M_Ret_Err := FALSE;
   S701_TL_LOCATE1_ERR.LP_Adv := FALSE;
   S701_TL_LOCATE1_ERR.LP_Ret := FALSE;
   S701_TL_LOCATE1_ERR.Visu_Adv := W#16#0;
   S701_TL_LOCATE1_ERR.Visu_Ret := W#16#0;
   S701_TL_LOCATE1_ERR.Error_T1.IN := FALSE;
   S701_TL_LOCATE1_ERR.Error_T1.PT := T#0MS;
   S701_TL_LOCATE1_ERR.Error_T1.Q := FALSE;
   S701_TL_LOCATE1_ERR.Error_T1.ET := T#0MS;
   S701_TL_LOCATE1_ERR.Error_T1.STATE := B#16#0;
   S701_TL_LOCATE1_ERR.Error_T1.STIME := T#0MS;
   S701_TL_LOCATE1_ERR.Error_T1.ATIME := T#0MS;
   S701_TL_LOCATE1_ERR.Error_T2.IN := FALSE;
   S701_TL_LOCATE1_ERR.Error_T2.PT := T#0MS;
   S701_TL_LOCATE1_ERR.Error_T2.Q := FALSE;
   S701_TL_LOCATE1_ERR.Error_T2.ET := T#0MS;
   S701_TL_LOCATE1_ERR.Error_T2.STATE := B#16#0;
   S701_TL_LOCATE1_ERR.Error_T2.STIME := T#0MS;
   S701_TL_LOCATE1_ERR.Error_T2.ATIME := T#0MS;
   S701_TL_LOCATE1_ERR.CHK_Aux1 := FALSE;
   S701_TL_LOCATE1_ERR.CHK_Aux2 := FALSE;
   S701_TL_LOCATE1_ERR.Error_T1_DN := FALSE;
   S701_TL_LOCATE1_ERR.Error_T2_DN := FALSE;
   S701_TL_LOCATE1_ERR.Adv_Memo := FALSE;
   S701_TL_LOCATE1_ERR.Visu_Adv_Arr[0] := FALSE;
   S701_TL_LOCATE1_ERR.Visu_Adv_Arr[1] := FALSE;
   S701_TL_LOCATE1_ERR.Visu_Adv_Arr[2] := FALSE;
   S701_TL_LOCATE1_ERR.Visu_Adv_Arr[3] := FALSE;
   S701_TL_LOCATE1_ERR.Visu_Adv_Arr[4] := FALSE;
   S701_TL_LOCATE1_ERR.Visu_Adv_Arr[5] := FALSE;
   S701_TL_LOCATE1_ERR.Visu_Adv_Arr[6] := FALSE;
   S701_TL_LOCATE1_ERR.Visu_Adv_Arr[7] := FALSE;
   S701_TL_LOCATE1_ERR.Visu_Adv_Arr[8] := FALSE;
   S701_TL_LOCATE1_ERR.Visu_Adv_Arr[9] := FALSE;
   S701_TL_LOCATE1_ERR.Visu_Adv_Arr[10] := FALSE;
   S701_TL_LOCATE1_ERR.Visu_Adv_Arr[11] := FALSE;
   S701_TL_LOCATE1_ERR.Visu_Adv_Arr[12] := FALSE;
   S701_TL_LOCATE1_ERR.Visu_Adv_Arr[13] := FALSE;
   S701_TL_LOCATE1_ERR.Visu_Adv_Arr[14] := FALSE;
